LIN {X 104.222,Y 43.174,Z 62.611,A 180.000,B 0.000,C 180.000} C_DIS
LIN {X 104.167,Y 43.026,Z 62.606,A 180.000,B 0.000,C 180.000} C_DIS
LIN {X 104.112,Y 42.878,Z 62.602,A 180.000,B 0.000,C 180.000} C_DIS
LIN {X 104.055,Y 42.732,Z 62.597,A 180.000,B 0.000,C 180.000} C_DIS
LIN {X 103.991,Y 42.588,Z 62.593,A 180.000,B 0.000,C 180.000} C_DIS
LIN {X 103.927,Y 42.444,Z 62.589,A 180.000,B 0.000,C 180.000} C_DIS
LIN {X 103.862,Y 42.300,Z 62.585,A 180.000,B 0.000,C 180.000} C_DIS
LIN {X 103.798,Y 42.156,Z 62.581,A 180.000,B 0.000,C 180.000} C_DIS
LIN {X 103.731,Y 42.014,Z 62.577,A 180.000,B 0.000,C 180.000} C_DIS
LIN {X 103.659,Y 41.874,Z 62.573,A 180.000,B 0.000,C 180.000} C_DIS
LIN {X 103.585,Y 41.735,Z 62.570,A 180.000,B 0.000,C 180.000} C_DIS
LIN {X 103.512,Y 41.595,Z 62.566,A 180.000,B 0.000,C 180.000} C_DIS
LIN {X 103.439,Y 41.456,Z 62.562,A 180.000,B 0.000,C 180.000} C_DIS
LIN {X 103.364,Y 41.317,Z 62.559,A 180.000,B 0.000,C 180.000} C_DIS
LIN {X 103.282,Y 41.183,Z 62.556,A 180.000,B 0.000,C 180.000} C_DIS
LIN {X 103.200,Y 41.048,Z 62.552,A 180.000,B 0.000,C 180.000} C_DIS
LIN {X 103.119,Y 40.913,Z 62.549,A 180.000,B 0.000,C 180.000} C_DIS
LIN {X 103.037,Y 40.779,Z 62.546,A 180.000,B 0.000,C 180.000} C_DIS
LIN {X 102.953,Y 40.646,Z 62.543,A 180.000,B 0.000,C 180.000} C_DIS
LIN {X 102.863,Y 40.516,Z 62.540,A 180.000,B 0.000,C 180.000} C_DIS
LIN {X 102.773,Y 40.387,Z 62.537,A 180.000,B 0.000,C 180.000} C_DIS
LIN {X 102.683,Y 40.258,Z 62.534,A 180.000,B 0.000,C 180.000} C_DIS
LIN {X 102.593,Y 40.128,Z 62.532,A 180.000,B 0.000,C 180.000} C_DIS
LIN {X 102.500,Y 40.001,Z 62.529,A 180.000,B 0.000,C 180.000} C_DIS
LIN {X 102.403,Y 39.878,Z 62.527,A 180.000,B 0.000,C 180.000} C_DIS
LIN {X 102.207,Y 39.631,Z 62.522,A 180.000,B 0.000,C 180.000} C_DIS
LIN {X 102.008,Y 39.386,Z 62.518,A 180.000,B 0.000,C 180.000} C_DIS
LIN {X 101.797,Y 39.152,Z 62.514,A 180.000,B 0.000,C 180.000} C_DIS
LIN {X 101.587,Y 38.918,Z 62.511,A 180.000,B 0.000,C 180.000} C_DIS
LIN {X 101.366,Y 38.694,Z 62.508,A 180.000,B 0.000,C 180.000} C_DIS
LIN {X 101.141,Y 38.473,Z 62.505,A 180.000,B 0.000,C 180.000} C_DIS
LIN {X 100.913,Y 38.256,Z 62.503,A 180.000,B 0.000,C 180.000} C_DIS
LIN {X 100.675,Y 38.050,Z 62.502,A 180.000,B 0.000,C 180.000} C_DIS
LIN {X 100.436,Y 37.844,Z 62.501,A 180.000,B 0.000,C 180.000} C_DIS
LIN {X 100.189,Y 37.649,Z 62.500,A 180.000,B 0.000,C 180.000} C_DIS
LIN {X 100.003,Y 37.508,Z 62.500,A 180.000,B 0.000,C 180.000} C_DIS
; Cutting Move Starts
LIN {X 99.815,Y 37.366,Z 62.500,A 180.000,B 0.000,C 180.000} C_DIS
LIN {X 99.757,Y 37.322,Z 62.500,A 180.000,B 0.000,C 180.000} C_DIS
LIN {X 99.578,Y 37.201,Z 62.500,A 180.000,B 0.000,C 180.000} C_DIS
LIN {X 99.221,Y 36.964,Z 62.500,A 180.000,B 0.000,C 180.000} C_DIS
LIN {X 99.042,Y 36.849,Z 62.500,A 180.000,B 0.000,C 180.000} C_DIS
LIN {X 99.009,Y 36.830,Z 62.500,A 180.000,B 0.000,C 180.000} C_DIS
LIN {X 98.505,Y 36.539,Z 62.500,A 180.000,B 0.000,C 180.000} C_DIS
LIN {X 98.385,Y 36.472,Z 62.500,A 180.000,B 0.000,C 180.000} C_DIS
LIN {X 98.327,Y 36.442,Z 62.500,A 180.000,B 0.000,C 180.000} C_DIS
LIN {X 97.790,Y 36.177,Z 62.500,A 180.000,B 0.000,C 180.000} C_DIS
LIN {X 97.659,Y 36.115,Z 62.500,A 180.000,B 0.000,C 180.000} C_DIS
LIN {X 97.612,Y 36.094,Z 62.500,A 180.000,B 0.000,C 180.000} C_DIS
LIN {X 97.075,Y 35.869,Z 62.500,A 180.000,B 0.000,C 180.000} C_DIS
LIN {X 96.897,Y 35.800,Z 62.500,A 180.000,B 0.000,C 180.000} C_DIS
LIN {X 96.360,Y 35.613,Z 62.500,A 180.000,B 0.000,C 180.000} C_DIS
LIN {X 96.258,Y 35.578,Z 62.500,A 180.000,B 0.000,C 180.000} C_DIS
LIN {X 96.181,Y 35.555,Z 62.500,A 180.000,B 0.000,C 180.000} C_DIS
LIN {X 96.003,Y 35.505,Z 62.500,A 180.000,B 0.000,C 180.000} C_DIS
LIN {X 95.625,Y 35.400,Z 62.500,A 180.000,B 0.000,C 180.000} C_DIS
LIN {X 95.466,Y 35.357,Z 62.500,A 180.000,B 0.000,C 180.000} C_DIS
LIN {X 95.288,Y 35.318,Z 62.500,A 180.000,B 0.000,C 180.000} C_DIS
LIN {X 94.828,Y 35.221,Z 62.500,A 180.000,B 0.000,C 180.000} C_DIS
LIN {X 94.751,Y 35.205,Z 62.500,A 180.000,B 0.000,C 180.000} C_DIS
LIN {X 94.573,Y 35.175,Z 62.500,A 180.000,B 0.000,C 180.000} C_DIS
LIN {X 94.036,Y 35.097,Z 62.500,A 180.000,B 0.000,C 180.000} C_DIS
LIN {X 93.857,Y 35.075,Z 62.500,A 180.000,B 0.000,C 180.000} C_DIS
LIN {X 93.679,Y 35.060,Z 62.500,A 180.000,B 0.000,C 180.000} C_DIS
LIN {X 93.321,Y 35.030,Z 62.500,A 180.000,B 0.000,C 180.000} C_DIS
LIN {X 93.142,Y 35.017,Z 62.500,A 180.000,B 0.000,C 180.000} C_DIS
LIN {X 92.964,Y 35.012,Z 62.500,A 180.000,B 0.000,C 180.000} C_DIS
LIN {X 92.606,Y 35.005,Z 62.500,A 180.000,B 0.000,C 180.000} C_DIS
LIN {X 92.427,Y 35.001,Z 62.500,A 180.000,B 0.000,C 180.000} C_DIS
LIN {X 92.249,Y 35.004,Z 62.500,A 180.000,B 0.000,C 180.000} C_DIS
LIN {X 91.712,Y 35.027,Z 62.500,A 180.000,B 0.000,C 180.000} C_DIS
LIN {X 91.533,Y 35.038,Z 62.500,A 180.000,B 0.000,C 180.000} C_DIS
LIN {X 91.489,Y 35.042,Z 62.500,A 180.000,B 0.000,C 180.000} C_DIS
LIN {X 90.997,Y 35.094,Z 62.500,A 180.000,B 0.000,C 180.000} C_DIS
LIN {X 90.818,Y 35.114,Z 62.500,A 180.000,B 0.000,C 180.000} C_DIS
LIN {X 90.640,Y 35.142,Z 62.500,A 180.000,B 0.000,C 180.000} C_DIS
LIN {X 90.103,Y 35.233,Z 62.500,A 180.000,B 0.000,C 180.000} C_DIS
LIN {X 89.925,Y 35.270,Z 62.500,A 180.000,B 0.000,C 180.000} C_DIS
LIN {X 89.372,Y 35.400,Z 62.500,A 180.000,B 0.000,C 180.000} C_DIS
LIN {X 89.209,Y 35.441,Z 62.500,A 180.000,B 0.000,C 180.000} C_DIS
LIN {X 89.031,Y 35.495,Z 62.500,A 180.000,B 0.000,C 180.000} C_DIS
LIN {X 88.673,Y 35.603,Z 62.500,A 180.000,B 0.000,C 180.000} C_DIS
LIN {X 88.494,Y 35.659,Z 62.500,A 180.000,B 0.000,C 180.000} C_DIS
LIN {X 45.590,Y 50.133,Z 62.500,A 180.000,B 0.000,C 180.000} C_DIS
LIN {X 45.411,Y 50.194,Z 62.500,A 180.000,B 0.000,C 180.000} C_DIS
LIN {X 45.296,Y 50.238,Z 62.500,A 180.000,B 0.000,C 180.000} C_DIS
LIN {X 45.232,Y 50.265,Z 62.500,A 180.000,B 0.000,C 180.000} C_DIS
LIN {X 45.053,Y 50.353,Z 62.500,A 180.000,B 0.000,C 180.000} C_DIS
LIN {X 44.944,Y 50.416,Z 62.500,A 180.000,B 0.000,C 180.000} C_DIS
LIN {X 44.874,Y 50.461,Z 62.500,A 180.000,B 0.000,C 180.000} C_DIS
LIN {X 44.785,Y 50.522,Z 62.500,A 180.000,B 0.000,C 180.000} C_DIS
LIN {X 44.696,Y 50.590,Z 62.500,A 180.000,B 0.000,C 180.000} C_DIS
LIN {X 44.689,Y 50.595,Z 62.500,A 180.000,B 0.000,C 180.000} C_DIS
LIN {X 44.603,Y 50.667,Z 62.500,A 180.000,B 0.000,C 180.000} C_DIS
LIN {X 44.517,Y 50.746,Z 62.500,A 180.000,B 0.000,C 180.000} C_DIS
LIN {X 44.488,Y 50.774,Z 62.500,A 180.000,B 0.000,C 180.000} C_DIS
LIN {X 44.410,Y 50.855,Z 62.500,A 180.000,B 0.000,C 180.000} C_DIS
LIN {X 44.338,Y 50.936,Z 62.500,A 180.000,B 0.000,C 180.000} C_DIS
LIN {X 44.325,Y 50.953,Z 62.500,A 180.000,B 0.000,C 180.000} C_DIS
LIN {X 44.254,Y 51.042,Z 62.500,A 180.000,B 0.000,C 180.000} C_DIS
LIN {X 44.189,Y 51.131,Z 62.500,A 180.000,B 0.000,C 180.000} C_DIS
LIN {X 44.159,Y 51.176,Z 62.500,A 180.000,B 0.000,C 180.000} C_DIS
LIN {X 44.077,Y 51.310,Z 62.500,A 180.000,B 0.000,C 180.000} C_DIS
LIN {X 43.984,Y 51.489,Z 62.500,A 180.000,B 0.000,C 180.000} C_DIS
LIN {X 43.981,Y 51.497,Z 62.500,A 180.000,B 0.000,C 180.000} C_DIS
LIN {X 43.909,Y 51.668,Z 62.500,A 180.000,B 0.000,C 180.000} C_DIS
LIN {X 43.849,Y 51.847,Z 62.500,A 180.000,B 0.000,C 180.000} C_DIS
LIN {X 43.804,Y 52.025,Z 62.500,A 180.000,B 0.000,C 180.000} C_DIS
LIN {X 43.802,Y 52.035,Z 62.500,A 180.000,B 0.000,C 180.000} C_DIS
LIN {X 43.772,Y 52.204,Z 62.500,A 180.000,B 0.000,C 180.000} C_DIS
LIN {X 43.754,Y 52.383,Z 62.500,A 180.000,B 0.000,C 180.000} C_DIS
LIN {X 43.748,Y 52.562,Z 62.500,A 180.000,B 0.000,C 180.000} C_DIS
LIN {X 43.756,Y 52.740,Z 62.500,A 180.000,B 0.000,C 180.000} C_DIS
LIN {X 43.776,Y 52.919,Z 62.500,A 180.000,B 0.000,C 180.000} C_DIS
LIN {X 43.802,Y 53.064,Z 62.500,A 180.000,B 0.000,C 180.000} C_DIS
LIN {X 43.809,Y 53.098,Z 62.500,A 180.000,B 0.000,C 180.000} C_DIS
LIN {X 43.856,Y 53.277,Z 62.500,A 180.000,B 0.000,C 180.000} C_DIS
LIN {X 43.916,Y 53.455,Z 62.500,A 180.000,B 0.000,C 180.000} C_DIS
LIN {X 50.248,Y 72.226,Z 62.500,A 180.000,B 0.000,C 180.000} C_DIS
LIN {X 50.311,Y 72.405,Z 62.500,A 180.000,B 0.000,C 180.000} C_DIS
LIN {X 50.388,Y 72.584,Z 62.500,A 180.000,B 0.000,C 180.000} C_DIS
LIN {X 50.416,Y 72.640,Z 62.500,A 180.000,B 0.000,C 180.000} C_DIS
LIN {X 50.484,Y 72.763,Z 62.500,A 180.000,B 0.000,C 180.000} C_DIS
LIN {X 50.595,Y 72.936,Z 62.500,A 180.000,B 0.000,C 180.000} C_DIS
LIN {X 50.599,Y 72.941,Z 62.500,A 180.000,B 0.000,C 180.000} C_DIS
LIN {X 50.665,Y 73.031,Z 62.500,A 180.000,B 0.000,C 180.000} C_DIS
LIN {X 50.737,Y 73.120,Z 62.500,A 180.000,B 0.000,C 180.000} C_DIS
LIN {X 50.774,Y 73.162,Z 62.500,A 180.000,B 0.000,C 180.000} C_DIS
LIN {X 50.905,Y 73.299,Z 62.500,A 180.000,B 0.000,C 180.000} C_DIS
LIN {X 50.953,Y 73.343,Z 62.500,A 180.000,B 0.000,C 180.000} C_DIS
LIN {X 51.112,Y 73.478,Z 62.500,A 180.000,B 0.000,C 180.000} C_DIS
LIN {X 51.131,Y 73.493,Z 62.500,A 180.000,B 0.000,C 180.000} C_DIS
LIN {X 51.310,Y 73.616,Z 62.500,A 180.000,B 0.000,C 180.000} C_DIS
LIN {X 51.376,Y 73.656,Z 62.500,A 180.000,B 0.000,C 180.000} C_DIS
LIN {X 51.489,Y 73.719,Z 62.500,A 180.000,B 0.000,C 180.000} C_DIS
LIN {X 51.668,Y 73.803,Z 62.500,A 180.000,B 0.000,C 180.000} C_DIS
LIN {X 51.749,Y 73.835,Z 62.500,A 180.000,B 0.000,C 180.000} C_DIS
LIN {X 51.847,Y 73.870,Z 62.500,A 180.000,B 0.000,C 180.000} C_DIS
LIN {X 52.025,Y 73.923,Z 62.500,A 180.000,B 0.000,C 180.000} C_DIS
LIN {X 52.204,Y 73.961,Z 62.500,A 180.000,B 0.000,C 180.000} C_DIS
LIN {X 52.383,Y 73.987,Z 62.500,A 180.000,B 0.000,C 180.000} C_DIS
LIN {X 52.562,Y 73.999,Z 62.500,A 180.000,B 0.000,C 180.000} C_DIS
LIN {X 52.740,Y 73.998,Z 62.500,A 180.000,B 0.000,C 180.000} C_DIS
LIN {X 52.919,Y 73.985,Z 62.500,A 180.000,B 0.000,C 180.000} C_DIS
LIN {X 53.098,Y 73.958,Z 62.500,A 180.000,B 0.000,C 180.000} C_DIS
LIN {X 53.277,Y 73.918,Z 62.500,A 180.000,B 0.000,C 180.000} C_DIS
LIN {X 53.455,Y 73.864,Z 62.500,A 180.000,B 0.000,C 180.000} C_DIS
LIN {X 83.198,Y 63.830,Z 62.500,A 180.000,B 0.000,C 180.000} C_DIS
LIN {X 96.464,Y 59.355,Z 62.500,A 180.000,B 0.000,C 180.000} C_DIS
LIN {X 96.539,Y 59.329,Z 62.500,A 180.000,B 0.000,C 180.000} C_DIS
LIN {X 96.718,Y 59.263,Z 62.500,A 180.000,B 0.000,C 180.000} C_DIS
LIN {X 97.075,Y 59.129,Z 62.500,A 180.000,B 0.000,C 180.000} C_DIS
LIN {X 97.254,Y 59.061,Z 62.500,A 180.000,B 0.000,C 180.000} C_DIS
LIN {X 97.397,Y 58.997,Z 62.500,A 180.000,B 0.000,C 180.000} C_DIS
LIN {X 97.798,Y 58.819,Z 62.500,A 180.000,B 0.000,C 180.000} C_DIS
LIN {X 97.969,Y 58.740,Z 62.500,A 180.000,B 0.000,C 180.000} C_DIS
LIN {X 98.148,Y 58.647,Z 62.500,A 180.000,B 0.000,C 180.000} C_DIS
LIN {X 98.505,Y 58.460,Z 62.500,A 180.000,B 0.000,C 180.000} C_DIS
LIN {X 98.684,Y 58.363,Z 62.500,A 180.000,B 0.000,C 180.000} C_DIS
LIN {X 98.817,Y 58.282,Z 62.500,A 180.000,B 0.000,C 180.000} C_DIS
LIN {X 99.221,Y 58.038,Z 62.500,A 180.000,B 0.000,C 180.000} C_DIS
LIN {X 99.395,Y 57.925,Z 62.500,A 180.000,B 0.000,C 180.000} C_DIS
LIN {X 99.757,Y 57.673,Z 62.500,A 180.000,B 0.000,C 180.000} C_DIS
LIN {X 99.909,Y 57.567,Z 62.500,A 180.000,B 0.000,C 180.000} C_DIS
LIN {X 99.936,Y 57.548,Z 62.500,A 180.000,B 0.000,C 180.000} C_DIS
LIN {X 100.114,Y 57.409,Z 62.500,A 180.000,B 0.000,C 180.000} C_DIS
LIN {X 100.472,Y 57.125,Z 62.500,A 180.000,B 0.000,C 180.000} C_DIS
LIN {X 100.588,Y 57.031,Z 62.500,A 180.000,B 0.000,C 180.000} C_DIS
LIN {X 100.651,Y 56.975,Z 62.500,A 180.000,B 0.000,C 180.000} C_DIS
LIN {X 101.008,Y 56.653,Z 62.500,A 180.000,B 0.000,C 180.000} C_DIS
LIN {X 101.180,Y 56.495,Z 62.500,A 180.000,B 0.000,C 180.000} C_DIS
LIN {X 101.187,Y 56.488,Z 62.500,A 180.000,B 0.000,C 180.000} C_DIS
LIN {X 101.356,Y 56.316,Z 62.500,A 180.000,B 0.000,C 180.000} C_DIS
LIN {X 101.545,Y 56.123,Z 62.500,A 180.000,B 0.000,C 180.000} C_DIS
LIN {X 101.704,Y 55.958,Z 62.500,A 180.000,B 0.000,C 180.000} C_DIS
LIN {X 101.723,Y 55.937,Z 62.500,A 180.000,B 0.000,C 180.000} C_DIS
LIN {X 101.860,Y 55.779,Z 62.500,A 180.000,B 0.000,C 180.000} C_DIS
LIN {X 102.168,Y 55.422,Z 62.500,A 180.000,B 0.000,C 180.000} C_DIS
LIN {X 102.260,Y 55.309,Z 62.500,A 180.000,B 0.000,C 180.000} C_DIS
LIN {X 102.310,Y 55.243,Z 62.500,A 180.000,B 0.000,C 180.000} C_DIS
LIN {X 102.617,Y 54.837,Z 62.500,A 180.000,B 0.000,C 180.000} C_DIS
LIN {X 102.713,Y 54.707,Z 62.500,A 180.000,B 0.000,C 180.000} C_DIS
LIN {X 102.796,Y 54.583,Z 62.500,A 180.000,B 0.000,C 180.000} C_DIS
LIN {X 103.069,Y 54.171,Z 62.500,A 180.000,B 0.000,C 180.000} C_DIS
LIN {X 103.153,Y 54.038,Z 62.500,A 180.000,B 0.000,C 180.000} C_DIS
LIN {X 103.180,Y 53.992,Z 62.500,A 180.000,B 0.000,C 180.000} C_DIS
LIN {X 103.386,Y 53.634,Z 62.500,A 180.000,B 0.000,C 180.000} C_DIS
LIN {X 103.489,Y 53.455,Z 62.500,A 180.000,B 0.000,C 180.000} C_DIS
LIN {X 103.511,Y 53.417,Z 62.500,A 180.000,B 0.000,C 180.000} C_DIS
LIN {X 103.583,Y 53.277,Z 62.500,A 180.000,B 0.000,C 180.000} C_DIS
LIN {X 103.760,Y 52.919,Z 62.500,A 180.000,B 0.000,C 180.000} C_DIS
LIN {X 103.848,Y 52.740,Z 62.500,A 180.000,B 0.000,C 180.000} C_DIS
LIN {X 103.869,Y 52.697,Z 62.500,A 180.000,B 0.000,C 180.000} C_DIS
LIN {X 103.927,Y 52.562,Z 62.500,A 180.000,B 0.000,C 180.000} C_DIS
LIN {X 104.077,Y 52.204,Z 62.500,A 180.000,B 0.000,C 180.000} C_DIS
LIN {X 104.152,Y 52.025,Z 62.500,A 180.000,B 0.000,C 180.000} C_DIS
LIN {X 104.218,Y 51.847,Z 62.500,A 180.000,B 0.000,C 180.000} C_DIS
LIN {X 104.405,Y 51.307,Z 62.500,A 180.000,B 0.000,C 180.000} C_DIS
LIN {X 104.459,Y 51.131,Z 62.500,A 180.000,B 0.000,C 180.000} C_DIS
LIN {X 104.609,Y 50.595,Z 62.500,A 180.000,B 0.000,C 180.000} C_DIS
LIN {X 104.654,Y 50.416,Z 62.500,A 180.000,B 0.000,C 180.000} C_DIS
LIN {X 104.692,Y 50.238,Z 62.500,A 180.000,B 0.000,C 180.000} C_DIS
LIN {X 104.768,Y 49.880,Z 62.500,A 180.000,B 0.000,C 180.000} C_DIS
LIN {X 104.805,Y 49.701,Z 62.500,A 180.000,B 0.000,C 180.000} C_DIS
LIN {X 104.832,Y 49.523,Z 62.500,A 180.000,B 0.000,C 180.000} C_DIS
LIN {X 104.885,Y 49.165,Z 62.500,A 180.000,B 0.000,C 180.000} C_DIS
LIN {X 104.911,Y 48.986,Z 62.500,A 180.000,B 0.000,C 180.000} C_DIS
LIN {X 104.929,Y 48.807,Z 62.500,A 180.000,B 0.000,C 180.000} C_DIS
LIN {X 104.974,Y 48.271,Z 62.500,A 180.000,B 0.000,C 180.000} C_DIS
LIN {X 104.986,Y 48.092,Z 62.500,A 180.000,B 0.000,C 180.000} C_DIS
LIN {X 104.989,Y 47.914,Z 62.500,A 180.000,B 0.000,C 180.000} C_DIS
LIN {X 104.996,Y 47.556,Z 62.500,A 180.000,B 0.000,C 180.000} C_DIS
LIN {X 104.999,Y 47.377,Z 62.500,A 180.000,B 0.000,C 180.000} C_DIS
LIN {X 104.994,Y 47.198,Z 62.500,A 180.000,B 0.000,C 180.000} C_DIS
LIN {X 104.971,Y 46.662,Z 62.500,A 180.000,B 0.000,C 180.000} C_DIS
LIN {X 104.957,Y 46.483,Z 62.500,A 180.000,B 0.000,C 180.000} C_DIS
LIN {X 104.900,Y 45.947,Z 62.500,A 180.000,B 0.000,C 180.000} C_DIS
LIN {X 104.879,Y 45.768,Z 62.500,A 180.000,B 0.000,C 180.000} C_DIS
LIN {X 104.850,Y 45.590,Z 62.500,A 180.000,B 0.000,C 180.000} C_DIS
LIN {X 104.789,Y 45.232,Z 62.500,A 180.000,B 0.000,C 180.000} C_DIS
LIN {X 104.762,Y 45.077,Z 62.500,A 180.000,B 0.000,C 180.000} C_DIS
LIN {X 104.758,Y 45.053,Z 62.500,A 180.000,B 0.000,C 180.000} C_DIS
LIN {X 104.719,Y 44.874,Z 62.500,A 180.000,B 0.000,C 180.000} C_DIS
LIN {X 104.592,Y 44.338,Z 62.500,A 180.000,B 0.000,C 180.000} C_DIS
LIN {X 104.584,Y 44.302,Z 62.500,A 180.000,B 0.000,C 180.000} C_DIS
LIN {X 104.544,Y 44.159,Z 62.500,A 180.000,B 0.000,C 180.000} C_DIS
LIN {X 104.381,Y 43.623,Z 62.500,A 180.000,B 0.000,C 180.000} C_DIS
LIN {X 104.323,Y 43.444,Z 62.500,A 180.000,B 0.000,C 180.000} C_DIS
LIN {X 104.257,Y 43.266,Z 62.500,A 180.000,B 0.000,C 180.000} C_DIS
LIN {X 104.123,Y 42.908,Z 62.500,A 180.000,B 0.000,C 180.000} C_DIS
LIN {X 104.053,Y 42.729,Z 62.500,A 180.000,B 0.000,C 180.000} C_DIS
LIN {X 104.047,Y 42.715,Z 62.500,A 180.000,B 0.000,C 180.000} C_DIS
LIN {X 103.974,Y 42.550,Z 62.500,A 180.000,B 0.000,C 180.000} C_DIS
LIN {X 103.814,Y 42.193,Z 62.500,A 180.000,B 0.000,C 180.000} C_DIS
LIN {X 103.732,Y 42.014,Z 62.500,A 180.000,B 0.000,C 180.000} C_DIS
LIN {X 103.690,Y 41.934,Z 62.500,A 180.000,B 0.000,C 180.000} C_DIS
LIN {X 103.451,Y 41.478,Z 62.500,A 180.000,B 0.000,C 180.000} C_DIS
LIN {X 103.353,Y 41.299,Z 62.500,A 180.000,B 0.000,C 180.000} C_DIS
LIN {X 103.332,Y 41.265,Z 62.500,A 180.000,B 0.000,C 180.000} C_DIS
LIN {X 103.027,Y 40.763,Z 62.500,A 180.000,B 0.000,C 180.000} C_DIS
LIN {X 102.975,Y 40.679,Z 62.500,A 180.000,B 0.000,C 180.000} C_DIS
LIN {X 102.910,Y 40.584,Z 62.500,A 180.000,B 0.000,C 180.000} C_DIS
LIN {X 102.617,Y 40.163,Z 62.500,A 180.000,B 0.000,C 180.000} C_DIS
LIN {X 102.536,Y 40.048,Z 62.500,A 180.000,B 0.000,C 180.000} C_DIS
LIN {X 102.438,Y 39.923,Z 62.500,A 180.000,B 0.000,C 180.000} C_DIS
LIN {X 102.112,Y 39.511,Z 62.500,A 180.000,B 0.000,C 180.000} C_DIS
LIN {X 102.081,Y 39.472,Z 62.500,A 180.000,B 0.000,C 180.000} C_DIS
LIN {X 101.960,Y 39.333,Z 62.500,A 180.000,B 0.000,C 180.000} C_DIS
LIN {X 101.638,Y 38.975,Z 62.500,A 180.000,B 0.000,C 180.000} C_DIS
LIN {X 101.545,Y 38.872,Z 62.500,A 180.000,B 0.000,C 180.000} C_DIS
LIN {X 101.471,Y 38.796,Z 62.500,A 180.000,B 0.000,C 180.000} C_DIS
LIN {X 101.366,Y 38.693,Z 62.500,A 180.000,B 0.000,C 180.000} C_DIS
LIN {X 101.008,Y 38.344,Z 62.500,A 180.000,B 0.000,C 180.000} C_DIS
LIN {X 100.918,Y 38.260,Z 62.500,A 180.000,B 0.000,C 180.000} C_DIS
LIN {X 100.829,Y 38.183,Z 62.500,A 180.000,B 0.000,C 180.000} C_DIS
LIN {X 100.472,Y 37.875,Z 62.500,A 180.000,B 0.000,C 180.000} C_DIS
LIN {X 100.293,Y 37.728,Z 62.500,A 180.000,B 0.000,C 180.000} C_DIS
LIN {X 100.003,Y 37.508,Z 62.500,A 180.000,B 0.000,C 180.000} C_DIS
; Link Move Starts
LIN {X 99.752,Y 37.319,Z 62.500,A 180.000,B 0.000,C 180.000} C_DIS
LIN {X 99.490,Y 37.143,Z 62.498,A 180.000,B 0.000,C 180.000} C_DIS
LIN {X 99.228,Y 36.969,Z 62.496,A 180.000,B 0.000,C 180.000} C_DIS
LIN {X 98.961,Y 36.802,Z 62.492,A 180.000,B 0.000,C 180.000} C_DIS
LIN {X 98.688,Y 36.645,Z 62.488,A 180.000,B 0.000,C 180.000} C_DIS
LIN {X 98.415,Y 36.488,Z 62.483,A 180.000,B 0.000,C 180.000} C_DIS
LIN {X 98.274,Y 36.416,Z 62.481,A 180.000,B 0.000,C 180.000} C_DIS
LIN {X 98.133,Y 36.346,Z 62.478,A 180.000,B 0.000,C 180.000} C_DIS
LIN {X 97.992,Y 36.276,Z 62.475,A 180.000,B 0.000,C 180.000} C_DIS
LIN {X 97.851,Y 36.207,Z 62.471,A 180.000,B 0.000,C 180.000} C_DIS
LIN {X 97.709,Y 36.137,Z 62.468,A 180.000,B 0.000,C 180.000} C_DIS
LIN {X 97.565,Y 36.075,Z 62.464,A 180.000,B 0.000,C 180.000} C_DIS
LIN {X 97.420,Y 36.014,Z 62.460,A 180.000,B 0.000,C 180.000} C_DIS
LIN {X 97.274,Y 35.953,Z 62.456,A 180.000,B 0.000,C 180.000} C_DIS
LIN {X 97.129,Y 35.892,Z 62.452,A 180.000,B 0.000,C 180.000} C_DIS
LIN {X 96.984,Y 35.832,Z 62.448,A 180.000,B 0.000,C 180.000} C_DIS
LIN {X 96.835,Y 35.779,Z 62.444,A 180.000,B 0.000,C 180.000} C_DIS
LIN {X 96.687,Y 35.727,Z 62.439,A 180.000,B 0.000,C 180.000} C_DIS
LIN {X 96.538,Y 35.675,Z 62.434,A 180.000,B 0.000,C 180.000} C_DIS
LIN {X 96.389,Y 35.623,Z 62.429,A 180.000,B 0.000,C 180.000} C_DIS
LIN {X 96.240,Y 35.573,Z 62.424,A 180.000,B 0.000,C 180.000} C_DIS
LIN {X 96.165,Y 35.550,Z 62.422,A 180.000,B 0.000,C 180.000} C_DIS
LIN {X 96.089,Y 35.529,Z 62.419,A 180.000,B 0.000,C 180.000} C_DIS
LIN {X 96.013,Y 35.508,Z 62.417,A 180.000,B 0.000,C 180.000} C_DIS
LIN {X 95.937,Y 35.487,Z 62.414,A 180.000,B 0.000,C 180.000} C_DIS
LIN {X 95.861,Y 35.465,Z 62.411,A 180.000,B 0.000,C 180.000} C_DIS
LIN {X 95.785,Y 35.444,Z 62.409,A 180.000,B 0.000,C 180.000} C_DIS
LIN {X 95.709,Y 35.423,Z 62.406,A 180.000,B 0.000,C 180.000} C_DIS
LIN {X 95.634,Y 35.402,Z 62.403,A 180.000,B 0.000,C 180.000} C_DIS
LIN {X 95.558,Y 35.381,Z 62.401,A 180.000,B 0.000,C 180.000} C_DIS
LIN {X 95.482,Y 35.361,Z 62.398,A 180.000,B 0.000,C 180.000} C_DIS
LIN {X 95.405,Y 35.343,Z 62.395,A 180.000,B 0.000,C 180.000} C_DIS
LIN {X 95.328,Y 35.327,Z 62.392,A 180.000,B 0.000,C 180.000} C_DIS
LIN {X 95.251,Y 35.310,Z 62.389,A 180.000,B 0.000,C 180.000} C_DIS
LIN {X 95.174,Y 35.294,Z 62.387,A 180.000,B 0.000,C 180.000} C_DIS
LIN {X 95.097,Y 35.278,Z 62.384,A 180.000,B 0.000,C 180.000} C_DIS
LIN {X 95.020,Y 35.261,Z 62.381,A 180.000,B 0.000,C 180.000} C_DIS
LIN {X 94.943,Y 35.245,Z 62.378,A 180.000,B 0.000,C 180.000} C_DIS
LIN {X 94.866,Y 35.229,Z 62.376,A 180.000,B 0.000,C 180.000} C_DIS
LIN {X 94.788,Y 35.212,Z 62.373,A 180.000,B 0.000,C 180.000} C_DIS
LIN {X 94.711,Y 35.197,Z 62.370,A 180.000,B 0.000,C 180.000} C_DIS
LIN {X 94.634,Y 35.184,Z 62.367,A 180.000,B 0.000,C 180.000} C_DIS
LIN {X 94.556,Y 35.173,Z 62.365,A 180.000,B 0.000,C 180.000} C_DIS
LIN {X 94.478,Y 35.161,Z 62.362,A 180.000,B 0.000,C 180.000} C_DIS
LIN {X 94.322,Y 35.138,Z 62.356,A 180.000,B 0.000,C 180.000} C_DIS
LIN {X 94.244,Y 35.127,Z 62.354,A 180.000,B 0.000,C 180.000} C_DIS
LIN {X 94.088,Y 35.104,Z 62.348,A 180.000,B 0.000,C 180.000} C_DIS
LIN {X 94.010,Y 35.093,Z 62.345,A 180.000,B 0.000,C 180.000} C_DIS
LIN {X 93.932,Y 35.082,Z 62.343,A 180.000,B 0.000,C 180.000} C_DIS
LIN {X 93.854,Y 35.074,Z 62.340,A 180.000,B 0.000,C 180.000} C_DIS
LIN {X 93.697,Y 35.061,Z 62.334,A 180.000,B 0.000,C 180.000} C_DIS
LIN {X 93.618,Y 35.055,Z 62.332,A 180.000,B 0.000,C 180.000} C_DIS
LIN {X 93.461,Y 35.042,Z 62.326,A 180.000,B 0.000,C 180.000} C_DIS
LIN {X 93.226,Y 35.022,Z 62.318,A 180.000,B 0.000,C 180.000} C_DIS
LIN {X 93.147,Y 35.017,Z 62.315,A 180.000,B 0.000,C 180.000} C_DIS
LIN {X 93.069,Y 35.014,Z 62.312,A 180.000,B 0.000,C 180.000} C_DIS
LIN {X 92.990,Y 35.012,Z 62.310,A 180.000,B 0.000,C 180.000} C_DIS
LIN {X 92.832,Y 35.009,Z 62.304,A 180.000,B 0.000,C 180.000} C_DIS
LIN {X 92.439,Y 35.001,Z 62.290,A 180.000,B 0.000,C 180.000} C_DIS
LIN {X 92.360,Y 35.001,Z 62.288,A 180.000,B 0.000,C 180.000} C_DIS
LIN {X 92.281,Y 35.003,Z 62.285,A 180.000,B 0.000,C 180.000} C_DIS
LIN {X 91.809,Y 35.023,Z 62.268,A 180.000,B 0.000,C 180.000} C_DIS
LIN {X 91.652,Y 35.030,Z 62.263,A 180.000,B 0.000,C 180.000} C_DIS
LIN {X 91.573,Y 35.034,Z 62.260,A 180.000,B 0.000,C 180.000} C_DIS
LIN {X 91.495,Y 35.042,Z 62.257,A 180.000,B 0.000,C 180.000} C_DIS
LIN {X 90.868,Y 35.108,Z 62.235,A 180.000,B 0.000,C 180.000} C_DIS
LIN {X 90.790,Y 35.117,Z 62.233,A 180.000,B 0.000,C 180.000} C_DIS
LIN {X 90.712,Y 35.130,Z 62.230,A 180.000,B 0.000,C 180.000} C_DIS
LIN {X 90.091,Y 35.235,Z 62.208,A 180.000,B 0.000,C 180.000} C_DIS
LIN {X 90.014,Y 35.250,Z 62.205,A 180.000,B 0.000,C 180.000} C_DIS
LIN {X 89.937,Y 35.267,Z 62.202,A 180.000,B 0.000,C 180.000} C_DIS
LIN {X 89.860,Y 35.285,Z 62.200,A 180.000,B 0.000,C 180.000} C_DIS
LIN {X 89.707,Y 35.321,Z 62.194,A 180.000,B 0.000,C 180.000} C_DIS
LIN {X 89.400,Y 35.393,Z 62.183,A 180.000,B 0.000,C 180.000} C_DIS
LIN {X 89.324,Y 35.411,Z 62.180,A 180.000,B 0.000,C 180.000} C_DIS
LIN {X 89.247,Y 35.431,Z 62.178,A 180.000,B 0.000,C 180.000} C_DIS
LIN {X 89.172,Y 35.452,Z 62.175,A 180.000,B 0.000,C 180.000} C_DIS
LIN {X 89.021,Y 35.498,Z 62.169,A 180.000,B 0.000,C 180.000} C_DIS
LIN {X 88.946,Y 35.521,Z 62.167,A 180.000,B 0.000,C 180.000} C_DIS
LIN {X 88.795,Y 35.567,Z 62.161,A 180.000,B 0.000,C 180.000} C_DIS
LIN {X 88.644,Y 35.612,Z 62.156,A 180.000,B 0.000,C 180.000} C_DIS
LIN {X 88.569,Y 35.635,Z 62.153,A 180.000,B 0.000,C 180.000} C_DIS
LIN {X 88.494,Y 35.659,Z 62.150,A 180.000,B 0.000,C 180.000} C_DIS
LIN {X 88.345,Y 35.710,Z 62.145,A 180.000,B 0.000,C 180.000} C_DIS
LIN {X 88.195,Y 35.760,Z 62.139,A 180.000,B 0.000,C 180.000} C_DIS
LIN {X 88.121,Y 35.785,Z 62.136,A 180.000,B 0.000,C 180.000} C_DIS
LIN {X 88.046,Y 35.810,Z 62.134,A 180.000,B 0.000,C 180.000} C_DIS
LIN {X 87.972,Y 35.836,Z 62.131,A 180.000,B 0.000,C 180.000} C_DIS
LIN {X 87.897,Y 35.861,Z 62.128,A 180.000,B 0.000,C 180.000} C_DIS
LIN {X 87.822,Y 35.886,Z 62.125,A 180.000,B 0.000,C 180.000} C_DIS
LIN {X 87.748,Y 35.911,Z 62.123,A 180.000,B 0.000,C 180.000} C_DIS
LIN {X 87.673,Y 35.936,Z 62.120,A 180.000,B 0.000,C 180.000} C_DIS
LIN {X 87.598,Y 35.961,Z 62.117,A 180.000,B 0.000,C 180.000} C_DIS
LIN {X 87.524,Y 35.987,Z 62.114,A 180.000,B 0.000,C 180.000} C_DIS
LIN {X 87.449,Y 36.012,Z 62.112,A 180.000,B 0.000,C 180.000} C_DIS
LIN {X 87.375,Y 36.037,Z 62.109,A 180.000,B 0.000,C 180.000} C_DIS
LIN {X 87.300,Y 36.062,Z 62.106,A 180.000,B 0.000,C 180.000} C_DIS
LIN {X 87.225,Y 36.087,Z 62.103,A 180.000,B 0.000,C 180.000} C_DIS
LIN {X 87.151,Y 36.112,Z 62.101,A 180.000,B 0.000,C 180.000} C_DIS
LIN {X 87.076,Y 36.138,Z 62.098,A 180.000,B 0.000,C 180.000} C_DIS
LIN {X 87.002,Y 36.163,Z 62.095,A 180.000,B 0.000,C 180.000} C_DIS
LIN {X 86.927,Y 36.188,Z 62.092,A 180.000,B 0.000,C 180.000} C_DIS
LIN {X 86.852,Y 36.213,Z 62.090,A 180.000,B 0.000,C 180.000} C_DIS
LIN {X 86.778,Y 36.238,Z 62.087,A 180.000,B 0.000,C 180.000} C_DIS
LIN {X 86.703,Y 36.263,Z 62.084,A 180.000,B 0.000,C 180.000} C_DIS
LIN {X 86.628,Y 36.289,Z 62.082,A 180.000,B 0.000,C 180.000} C_DIS
LIN {X 86.554,Y 36.314,Z 62.079,A 180.000,B 0.000,C 180.000} C_DIS
LIN {X 86.479,Y 36.339,Z 62.077,A 180.000,B 0.000,C 180.000} C_DIS
LIN {X 86.405,Y 36.364,Z 62.074,A 180.000,B 0.000,C 180.000} C_DIS
LIN {X 86.255,Y 36.415,Z 62.069,A 180.000,B 0.000,C 180.000} C_DIS
LIN {X 86.106,Y 36.465,Z 62.064,A 180.000,B 0.000,C 180.000} C_DIS
LIN {X 85.957,Y 36.515,Z 62.060,A 180.000,B 0.000,C 180.000} C_DIS
LIN {X 85.808,Y 36.566,Z 62.055,A 180.000,B 0.000,C 180.000} C_DIS
LIN {X 85.658,Y 36.616,Z 62.051,A 180.000,B 0.000,C 180.000} C_DIS
LIN {X 85.509,Y 36.666,Z 62.047,A 180.000,B 0.000,C 180.000} C_DIS
LIN {X 85.360,Y 36.717,Z 62.042,A 180.000,B 0.000,C 180.000} C_DIS
LIN {X 85.211,Y 36.767,Z 62.039,A 180.000,B 0.000,C 180.000} C_DIS
LIN {X 85.061,Y 36.817,Z 62.035,A 180.000,B 0.000,C 180.000} C_DIS
LIN {X 84.912,Y 36.868,Z 62.031,A 180.000,B 0.000,C 180.000} C_DIS
LIN {X 84.763,Y 36.918,Z 62.028,A 180.000,B 0.000,C 180.000} C_DIS
LIN {X 84.614,Y 36.968,Z 62.024,A 180.000,B 0.000,C 180.000} C_DIS
LIN {X 84.465,Y 37.019,Z 62.021,A 180.000,B 0.000,C 180.000} C_DIS
LIN {X 84.315,Y 37.069,Z 62.019,A 180.000,B 0.000,C 180.000} C_DIS
LIN {X 84.166,Y 37.119,Z 62.016,A 180.000,B 0.000,C 180.000} C_DIS
LIN {X 83.868,Y 37.220,Z 62.011,A 180.000,B 0.000,C 180.000} C_DIS
LIN {X 83.569,Y 37.321,Z 62.007,A 180.000,B 0.000,C 180.000} C_DIS
LIN {X 83.271,Y 37.421,Z 62.004,A 180.000,B 0.000,C 180.000} C_DIS
LIN {X 82.972,Y 37.522,Z 62.002,A 180.000,B 0.000,C 180.000} C_DIS
LIN {X 82.674,Y 37.623,Z 62.000,A 180.000,B 0.000,C 180.000} C_DIS
LIN {X 82.417,Y 37.709,Z 62.000,A 180.000,B 0.000,C 180.000} C_DIS
; Cutting Move Starts
LIN {X 45.590,Y 50.133,Z 62.000,A 180.000,B 0.000,C 180.000} C_DIS
LIN {X 45.411,Y 50.194,Z 62.000,A 180.000,B 0.000,C 180.000} C_DIS
LIN {X 45.296,Y 50.238,Z 62.000,A 180.000,B 0.000,C 180.000} C_DIS
LIN {X 45.232,Y 50.265,Z 62.000,A 180.000,B 0.000,C 180.000} C_DIS
LIN {X 45.053,Y 50.353,Z 62.000,A 180.000,B 0.000,C 180.000} C_DIS
LIN {X 44.944,Y 50.416,Z 62.000,A 180.000,B 0.000,C 180.000} C_DIS
LIN {X 44.874,Y 50.461,Z 62.000,A 180.000,B 0.000,C 180.000} C_DIS
LIN {X 44.785,Y 50.522,Z 62.000,A 180.000,B 0.000,C 180.000} C_DIS
LIN {X 44.696,Y 50.590,Z 62.000,A 180.000,B 0.000,C 180.000} C_DIS
LIN {X 44.689,Y 50.595,Z 62.000,A 180.000,B 0.000,C 180.000} C_DIS
LIN {X 44.603,Y 50.667,Z 62.000,A 180.000,B 0.000,C 180.000} C_DIS
LIN {X 44.517,Y 50.746,Z 62.000,A 180.000,B 0.000,C 180.000} C_DIS
LIN {X 44.488,Y 50.774,Z 62.000,A 180.000,B 0.000,C 180.000} C_DIS
LIN {X 44.410,Y 50.855,Z 62.000,A 180.000,B 0.000,C 180.000} C_DIS
LIN {X 44.338,Y 50.936,Z 62.000,A 180.000,B 0.000,C 180.000} C_DIS
LIN {X 44.325,Y 50.953,Z 62.000,A 180.000,B 0.000,C 180.000} C_DIS
LIN {X 44.254,Y 51.042,Z 62.000,A 180.000,B 0.000,C 180.000} C_DIS
LIN {X 44.189,Y 51.131,Z 62.000,A 180.000,B 0.000,C 180.000} C_DIS
LIN {X 44.159,Y 51.176,Z 62.000,A 180.000,B 0.000,C 180.000} C_DIS
LIN {X 44.077,Y 51.310,Z 62.000,A 180.000,B 0.000,C 180.000} C_DIS
LIN {X 43.984,Y 51.489,Z 62.000,A 180.000,B 0.000,C 180.000} C_DIS
LIN {X 43.981,Y 51.497,Z 62.000,A 180.000,B 0.000,C 180.000} C_DIS
LIN {X 43.909,Y 51.668,Z 62.000,A 180.000,B 0.000,C 180.000} C_DIS
LIN {X 43.849,Y 51.847,Z 62.000,A 180.000,B 0.000,C 180.000} C_DIS
LIN {X 43.804,Y 52.025,Z 62.000,A 180.000,B 0.000,C 180.000} C_DIS
LIN {X 43.802,Y 52.035,Z 62.000,A 180.000,B 0.000,C 180.000} C_DIS
LIN {X 43.772,Y 52.204,Z 62.000,A 180.000,B 0.000,C 180.000} C_DIS
LIN {X 43.754,Y 52.383,Z 62.000,A 180.000,B 0.000,C 180.000} C_DIS
LIN {X 43.748,Y 52.562,Z 62.000,A 180.000,B 0.000,C 180.000} C_DIS
LIN {X 43.756,Y 52.740,Z 62.000,A 180.000,B 0.000,C 180.000} C_DIS
LIN {X 43.776,Y 52.919,Z 62.000,A 180.000,B 0.000,C 180.000} C_DIS
LIN {X 43.802,Y 53.064,Z 62.000,A 180.000,B 0.000,C 180.000} C_DIS
LIN {X 43.809,Y 53.098,Z 62.000,A 180.000,B 0.000,C 180.000} C_DIS
LIN {X 43.856,Y 53.277,Z 62.000,A 180.000,B 0.000,C 180.000} C_DIS
LIN {X 43.916,Y 53.455,Z 62.000,A 180.000,B 0.000,C 180.000} C_DIS
LIN {X 50.248,Y 72.226,Z 62.000,A 180.000,B 0.000,C 180.000} C_DIS
LIN {X 50.311,Y 72.405,Z 62.000,A 180.000,B 0.000,C 180.000} C_DIS
LIN {X 50.388,Y 72.584,Z 62.000,A 180.000,B 0.000,C 180.000} C_DIS
LIN {X 50.416,Y 72.640,Z 62.000,A 180.000,B 0.000,C 180.000} C_DIS
LIN {X 50.484,Y 72.763,Z 62.000,A 180.000,B 0.000,C 180.000} C_DIS
LIN {X 50.595,Y 72.936,Z 62.000,A 180.000,B 0.000,C 180.000} C_DIS
LIN {X 50.599,Y 72.941,Z 62.000,A 180.000,B 0.000,C 180.000} C_DIS
LIN {X 50.665,Y 73.031,Z 62.000,A 180.000,B 0.000,C 180.000} C_DIS
LIN {X 50.737,Y 73.120,Z 62.000,A 180.000,B 0.000,C 180.000} C_DIS
LIN {X 50.774,Y 73.162,Z 62.000,A 180.000,B 0.000,C 180.000} C_DIS
LIN {X 50.905,Y 73.299,Z 62.000,A 180.000,B 0.000,C 180.000} C_DIS
LIN {X 50.953,Y 73.343,Z 62.000,A 180.000,B 0.000,C 180.000} C_DIS
LIN {X 51.112,Y 73.478,Z 62.000,A 180.000,B 0.000,C 180.000} C_DIS
LIN {X 51.131,Y 73.493,Z 62.000,A 180.000,B 0.000,C 180.000} C_DIS
LIN {X 51.310,Y 73.616,Z 62.000,A 180.000,B 0.000,C 180.000} C_DIS
LIN {X 51.376,Y 73.656,Z 62.000,A 180.000,B 0.000,C 180.000} C_DIS
LIN {X 51.489,Y 73.719,Z 62.000,A 180.000,B 0.000,C 180.000} C_DIS
LIN {X 51.668,Y 73.803,Z 62.000,A 180.000,B 0.000,C 180.000} C_DIS
LIN {X 51.749,Y 73.835,Z 62.000,A 180.000,B 0.000,C 180.000} C_DIS
LIN {X 51.847,Y 73.870,Z 62.000,A 180.000,B 0.000,C 180.000} C_DIS
LIN {X 52.025,Y 73.923,Z 62.000,A 180.000,B 0.000,C 180.000} C_DIS
LIN {X 52.204,Y 73.961,Z 62.000,A 180.000,B 0.000,C 180.000} C_DIS
LIN {X 52.383,Y 73.987,Z 62.000,A 180.000,B 0.000,C 180.000} C_DIS
LIN {X 52.562,Y 73.999,Z 62.000,A 180.000,B 0.000,C 180.000} C_DIS
LIN {X 52.740,Y 73.998,Z 62.000,A 180.000,B 0.000,C 180.000} C_DIS
LIN {X 52.919,Y 73.985,Z 62.000,A 180.000,B 0.000,C 180.000} C_DIS
LIN {X 53.098,Y 73.958,Z 62.000,A 180.000,B 0.000,C 180.000} C_DIS
LIN {X 53.277,Y 73.918,Z 62.000,A 180.000,B 0.000,C 180.000} C_DIS
LIN {X 53.455,Y 73.864,Z 62.000,A 180.000,B 0.000,C 180.000} C_DIS
LIN {X 83.198,Y 63.830,Z 62.000,A 180.000,B 0.000,C 180.000} C_DIS
LIN {X 96.464,Y 59.355,Z 62.000,A 180.000,B 0.000,C 180.000} C_DIS
LIN {X 96.539,Y 59.329,Z 62.000,A 180.000,B 0.000,C 180.000} C_DIS
LIN {X 96.718,Y 59.263,Z 62.000,A 180.000,B 0.000,C 180.000} C_DIS
LIN {X 97.075,Y 59.129,Z 62.000,A 180.000,B 0.000,C 180.000} C_DIS
LIN {X 97.254,Y 59.061,Z 62.000,A 180.000,B 0.000,C 180.000} C_DIS
LIN {X 97.397,Y 58.997,Z 62.000,A 180.000,B 0.000,C 180.000} C_DIS
LIN {X 97.798,Y 58.819,Z 62.000,A 180.000,B 0.000,C 180.000} C_DIS
LIN {X 97.969,Y 58.740,Z 62.000,A 180.000,B 0.000,C 180.000} C_DIS
LIN {X 98.148,Y 58.647,Z 62.000,A 180.000,B 0.000,C 180.000} C_DIS
LIN {X 98.505,Y 58.460,Z 62.000,A 180.000,B 0.000,C 180.000} C_DIS
LIN {X 98.684,Y 58.363,Z 62.000,A 180.000,B 0.000,C 180.000} C_DIS
LIN {X 98.817,Y 58.282,Z 62.000,A 180.000,B 0.000,C 180.000} C_DIS
LIN {X 99.221,Y 58.038,Z 62.000,A 180.000,B 0.000,C 180.000} C_DIS
LIN {X 99.395,Y 57.925,Z 62.000,A 180.000,B 0.000,C 180.000} C_DIS
LIN {X 99.757,Y 57.673,Z 62.000,A 180.000,B 0.000,C 180.000} C_DIS
LIN {X 99.909,Y 57.567,Z 62.000,A 180.000,B 0.000,C 180.000} C_DIS
LIN {X 99.936,Y 57.548,Z 62.000,A 180.000,B 0.000,C 180.000} C_DIS
LIN {X 100.114,Y 57.409,Z 62.000,A 180.000,B 0.000,C 180.000} C_DIS
LIN {X 100.472,Y 57.125,Z 62.000,A 180.000,B 0.000,C 180.000} C_DIS
LIN {X 100.588,Y 57.031,Z 62.000,A 180.000,B 0.000,C 180.000} C_DIS
LIN {X 100.651,Y 56.975,Z 62.000,A 180.000,B 0.000,C 180.000} C_DIS
LIN {X 101.008,Y 56.653,Z 62.000,A 180.000,B 0.000,C 180.000} C_DIS
LIN {X 101.180,Y 56.495,Z 62.000,A 180.000,B 0.000,C 180.000} C_DIS
LIN {X 101.187,Y 56.488,Z 62.000,A 180.000,B 0.000,C 180.000} C_DIS
LIN {X 101.356,Y 56.316,Z 62.000,A 180.000,B 0.000,C 180.000} C_DIS
LIN {X 101.545,Y 56.123,Z 62.000,A 180.000,B 0.000,C 180.000} C_DIS
LIN {X 101.704,Y 55.958,Z 62.000,A 180.000,B 0.000,C 180.000} C_DIS
LIN {X 101.723,Y 55.937,Z 62.000,A 180.000,B 0.000,C 180.000} C_DIS
LIN {X 101.860,Y 55.779,Z 62.000,A 180.000,B 0.000,C 180.000} C_DIS
LIN {X 102.168,Y 55.422,Z 62.000,A 180.000,B 0.000,C 180.000} C_DIS
LIN {X 102.260,Y 55.309,Z 62.000,A 180.000,B 0.000,C 180.000} C_DIS
LIN {X 102.310,Y 55.243,Z 62.000,A 180.000,B 0.000,C 180.000} C_DIS
LIN {X 102.617,Y 54.837,Z 62.000,A 180.000,B 0.000,C 180.000} C_DIS
LIN {X 102.713,Y 54.707,Z 62.000,A 180.000,B 0.000,C 180.000} C_DIS
LIN {X 102.796,Y 54.583,Z 62.000,A 180.000,B 0.000,C 180.000} C_DIS
LIN {X 103.069,Y 54.171,Z 62.000,A 180.000,B 0.000,C 180.000} C_DIS
LIN {X 103.153,Y 54.038,Z 62.000,A 180.000,B 0.000,C 180.000} C_DIS
LIN {X 103.180,Y 53.992,Z 62.000,A 180.000,B 0.000,C 180.000} C_DIS
LIN {X 103.386,Y 53.634,Z 62.000,A 180.000,B 0.000,C 180.000} C_DIS
LIN {X 103.489,Y 53.455,Z 62.000,A 180.000,B 0.000,C 180.000} C_DIS
LIN {X 103.511,Y 53.417,Z 62.000,A 180.000,B 0.000,C 180.000} C_DIS
LIN {X 103.583,Y 53.277,Z 62.000,A 180.000,B 0.000,C 180.000} C_DIS
LIN {X 103.760,Y 52.919,Z 62.000,A 180.000,B 0.000,C 180.000} C_DIS
LIN {X 103.848,Y 52.740,Z 62.000,A 180.000,B 0.000,C 180.000} C_DIS
LIN {X 103.869,Y 52.697,Z 62.000,A 180.000,B 0.000,C 180.000} C_DIS
LIN {X 103.927,Y 52.562,Z 62.000,A 180.000,B 0.000,C 180.000} C_DIS
LIN {X 104.077,Y 52.204,Z 62.000,A 180.000,B 0.000,C 180.000} C_DIS
LIN {X 104.152,Y 52.025,Z 62.000,A 180.000,B 0.000,C 180.000} C_DIS
LIN {X 104.218,Y 51.847,Z 62.000,A 180.000,B 0.000,C 180.000} C_DIS
LIN {X 104.405,Y 51.307,Z 62.000,A 180.000,B 0.000,C 180.000} C_DIS
LIN {X 104.459,Y 51.131,Z 62.000,A 180.000,B 0.000,C 180.000} C_DIS
LIN {X 104.609,Y 50.595,Z 62.000,A 180.000,B 0.000,C 180.000} C_DIS
LIN {X 104.654,Y 50.416,Z 62.000,A 180.000,B 0.000,C 180.000} C_DIS
LIN {X 104.692,Y 50.238,Z 62.000,A 180.000,B 0.000,C 180.000} C_DIS
LIN {X 104.768,Y 49.880,Z 62.000,A 180.000,B 0.000,C 180.000} C_DIS
LIN {X 104.805,Y 49.701,Z 62.000,A 180.000,B 0.000,C 180.000} C_DIS
LIN {X 104.832,Y 49.523,Z 62.000,A 180.000,B 0.000,C 180.000} C_DIS
LIN {X 104.885,Y 49.165,Z 62.000,A 180.000,B 0.000,C 180.000} C_DIS
LIN {X 104.911,Y 48.986,Z 62.000,A 180.000,B 0.000,C 180.000} C_DIS
LIN {X 104.929,Y 48.807,Z 62.000,A 180.000,B 0.000,C 180.000} C_DIS
LIN {X 104.974,Y 48.271,Z 62.000,A 180.000,B 0.000,C 180.000} C_DIS
LIN {X 104.986,Y 48.092,Z 62.000,A 180.000,B 0.000,C 180.000} C_DIS
LIN {X 104.989,Y 47.914,Z 62.000,A 180.000,B 0.000,C 180.000} C_DIS
LIN {X 104.996,Y 47.556,Z 62.000,A 180.000,B 0.000,C 180.000} C_DIS
LIN {X 104.999,Y 47.377,Z 62.000,A 180.000,B 0.000,C 180.000} C_DIS
LIN {X 104.994,Y 47.198,Z 62.000,A 180.000,B 0.000,C 180.000} C_DIS
LIN {X 104.971,Y 46.662,Z 62.000,A 180.000,B 0.000,C 180.000} C_DIS
LIN {X 104.957,Y 46.483,Z 62.000,A 180.000,B 0.000,C 180.000} C_DIS
LIN {X 104.900,Y 45.947,Z 62.000,A 180.000,B 0.000,C 180.000} C_DIS
LIN {X 104.879,Y 45.768,Z 62.000,A 180.000,B 0.000,C 180.000} C_DIS
LIN {X 104.850,Y 45.590,Z 62.000,A 180.000,B 0.000,C 180.000} C_DIS
LIN {X 104.789,Y 45.232,Z 62.000,A 180.000,B 0.000,C 180.000} C_DIS
LIN {X 104.762,Y 45.077,Z 62.000,A 180.000,B 0.000,C 180.000} C_DIS
LIN {X 104.758,Y 45.053,Z 62.000,A 180.000,B 0.000,C 180.000} C_DIS
LIN {X 104.719,Y 44.874,Z 62.000,A 180.000,B 0.000,C 180.000} C_DIS
LIN {X 104.592,Y 44.338,Z 62.000,A 180.000,B 0.000,C 180.000} C_DIS
LIN {X 104.584,Y 44.302,Z 62.000,A 180.000,B 0.000,C 180.000} C_DIS
LIN {X 104.544,Y 44.159,Z 62.000,A 180.000,B 0.000,C 180.000} C_DIS
LIN {X 104.381,Y 43.623,Z 62.000,A 180.000,B 0.000,C 180.000} C_DIS
LIN {X 104.323,Y 43.444,Z 62.000,A 180.000,B 0.000,C 180.000} C_DIS
LIN {X 104.257,Y 43.266,Z 62.000,A 180.000,B 0.000,C 180.000} C_DIS
LIN {X 104.123,Y 42.908,Z 62.000,A 180.000,B 0.000,C 180.000} C_DIS
LIN {X 104.053,Y 42.729,Z 62.000,A 180.000,B 0.000,C 180.000} C_DIS
LIN {X 104.047,Y 42.715,Z 62.000,A 180.000,B 0.000,C 180.000} C_DIS
LIN {X 103.974,Y 42.550,Z 62.000,A 180.000,B 0.000,C 180.000} C_DIS
LIN {X 103.814,Y 42.193,Z 62.000,A 180.000,B 0.000,C 180.000} C_DIS
LIN {X 103.732,Y 42.014,Z 62.000,A 180.000,B 0.000,C 180.000} C_DIS
LIN {X 103.690,Y 41.934,Z 62.000,A 180.000,B 0.000,C 180.000} C_DIS
LIN {X 103.451,Y 41.478,Z 62.000,A 180.000,B 0.000,C 180.000} C_DIS
LIN {X 103.353,Y 41.299,Z 62.000,A 180.000,B 0.000,C 180.000} C_DIS
LIN {X 103.332,Y 41.265,Z 62.000,A 180.000,B 0.000,C 180.000} C_DIS
LIN {X 103.027,Y 40.763,Z 62.000,A 180.000,B 0.000,C 180.000} C_DIS
LIN {X 102.975,Y 40.679,Z 62.000,A 180.000,B 0.000,C 180.000} C_DIS
LIN {X 102.910,Y 40.584,Z 62.000,A 180.000,B 0.000,C 180.000} C_DIS
LIN {X 102.617,Y 40.163,Z 62.000,A 180.000,B 0.000,C 180.000} C_DIS
LIN {X 102.536,Y 40.048,Z 62.000,A 180.000,B 0.000,C 180.000} C_DIS
LIN {X 102.438,Y 39.923,Z 62.000,A 180.000,B 0.000,C 180.000} C_DIS
LIN {X 102.112,Y 39.511,Z 62.000,A 180.000,B 0.000,C 180.000} C_DIS
LIN {X 102.081,Y 39.472,Z 62.000,A 180.000,B 0.000,C 180.000} C_DIS
LIN {X 101.960,Y 39.333,Z 62.000,A 180.000,B 0.000,C 180.000} C_DIS
LIN {X 101.638,Y 38.975,Z 62.000,A 180.000,B 0.000,C 180.000} C_DIS
LIN {X 101.545,Y 38.872,Z 62.000,A 180.000,B 0.000,C 180.000} C_DIS
LIN {X 101.471,Y 38.796,Z 62.000,A 180.000,B 0.000,C 180.000} C_DIS
LIN {X 101.366,Y 38.693,Z 62.000,A 180.000,B 0.000,C 180.000} C_DIS
LIN {X 101.008,Y 38.344,Z 62.000,A 180.000,B 0.000,C 180.000} C_DIS
LIN {X 100.918,Y 38.260,Z 62.000,A 180.000,B 0.000,C 180.000} C_DIS
LIN {X 100.829,Y 38.183,Z 62.000,A 180.000,B 0.000,C 180.000} C_DIS
LIN {X 100.472,Y 37.875,Z 62.000,A 180.000,B 0.000,C 180.000} C_DIS
LIN {X 100.293,Y 37.728,Z 62.000,A 180.000,B 0.000,C 180.000} C_DIS
LIN {X 100.003,Y 37.508,Z 62.000,A 180.000,B 0.000,C 180.000} C_DIS
LIN {X 99.815,Y 37.366,Z 62.000,A 180.000,B 0.000,C 180.000} C_DIS
LIN {X 99.757,Y 37.322,Z 62.000,A 180.000,B 0.000,C 180.000} C_DIS
LIN {X 99.578,Y 37.201,Z 62.000,A 180.000,B 0.000,C 180.000} C_DIS
LIN {X 99.221,Y 36.964,Z 62.000,A 180.000,B 0.000,C 180.000} C_DIS
LIN {X 99.042,Y 36.849,Z 62.000,A 180.000,B 0.000,C 180.000} C_DIS
LIN {X 99.009,Y 36.830,Z 62.000,A 180.000,B 0.000,C 180.000} C_DIS
LIN {X 98.505,Y 36.539,Z 62.000,A 180.000,B 0.000,C 180.000} C_DIS
LIN {X 98.385,Y 36.472,Z 62.000,A 180.000,B 0.000,C 180.000} C_DIS
LIN {X 98.327,Y 36.442,Z 62.000,A 180.000,B 0.000,C 180.000} C_DIS
LIN {X 97.790,Y 36.177,Z 62.000,A 180.000,B 0.000,C 180.000} C_DIS
LIN {X 97.659,Y 36.115,Z 62.000,A 180.000,B 0.000,C 180.000} C_DIS
LIN {X 97.612,Y 36.094,Z 62.000,A 180.000,B 0.000,C 180.000} C_DIS
LIN {X 97.075,Y 35.869,Z 62.000,A 180.000,B 0.000,C 180.000} C_DIS
LIN {X 96.897,Y 35.800,Z 62.000,A 180.000,B 0.000,C 180.000} C_DIS
LIN {X 96.360,Y 35.613,Z 62.000,A 180.000,B 0.000,C 180.000} C_DIS
LIN {X 96.258,Y 35.578,Z 62.000,A 180.000,B 0.000,C 180.000} C_DIS
LIN {X 96.181,Y 35.555,Z 62.000,A 180.000,B 0.000,C 180.000} C_DIS
LIN {X 96.003,Y 35.505,Z 62.000,A 180.000,B 0.000,C 180.000} C_DIS
LIN {X 95.625,Y 35.400,Z 62.000,A 180.000,B 0.000,C 180.000} C_DIS
LIN {X 95.466,Y 35.357,Z 62.000,A 180.000,B 0.000,C 180.000} C_DIS
LIN {X 95.288,Y 35.318,Z 62.000,A 180.000,B 0.000,C 180.000} C_DIS
LIN {X 94.828,Y 35.221,Z 62.000,A 180.000,B 0.000,C 180.000} C_DIS
LIN {X 94.751,Y 35.205,Z 62.000,A 180.000,B 0.000,C 180.000} C_DIS
LIN {X 94.573,Y 35.175,Z 62.000,A 180.000,B 0.000,C 180.000} C_DIS
LIN {X 94.036,Y 35.097,Z 62.000,A 180.000,B 0.000,C 180.000} C_DIS
LIN {X 93.857,Y 35.075,Z 62.000,A 180.000,B 0.000,C 180.000} C_DIS
LIN {X 93.679,Y 35.060,Z 62.000,A 180.000,B 0.000,C 180.000} C_DIS
LIN {X 93.321,Y 35.030,Z 62.000,A 180.000,B 0.000,C 180.000} C_DIS
LIN {X 93.142,Y 35.017,Z 62.000,A 180.000,B 0.000,C 180.000} C_DIS
LIN {X 92.964,Y 35.012,Z 62.000,A 180.000,B 0.000,C 180.000} C_DIS
LIN {X 92.606,Y 35.005,Z 62.000,A 180.000,B 0.000,C 180.000} C_DIS
LIN {X 92.427,Y 35.001,Z 62.000,A 180.000,B 0.000,C 180.000} C_DIS
LIN {X 92.249,Y 35.004,Z 62.000,A 180.000,B 0.000,C 180.000} C_DIS
LIN {X 91.712,Y 35.027,Z 62.000,A 180.000,B 0.000,C 180.000} C_DIS
LIN {X 91.533,Y 35.038,Z 62.000,A 180.000,B 0.000,C 180.000} C_DIS
LIN {X 91.489,Y 35.042,Z 62.000,A 180.000,B 0.000,C 180.000} C_DIS
LIN {X 90.997,Y 35.094,Z 62.000,A 180.000,B 0.000,C 180.000} C_DIS
LIN {X 90.818,Y 35.114,Z 62.000,A 180.000,B 0.000,C 180.000} C_DIS
LIN {X 90.640,Y 35.142,Z 62.000,A 180.000,B 0.000,C 180.000} C_DIS
LIN {X 90.103,Y 35.233,Z 62.000,A 180.000,B 0.000,C 180.000} C_DIS
LIN {X 89.925,Y 35.270,Z 62.000,A 180.000,B 0.000,C 180.000} C_DIS
LIN {X 89.372,Y 35.400,Z 62.000,A 180.000,B 0.000,C 180.000} C_DIS
LIN {X 89.209,Y 35.441,Z 62.000,A 180.000,B 0.000,C 180.000} C_DIS
LIN {X 89.031,Y 35.495,Z 62.000,A 180.000,B 0.000,C 180.000} C_DIS
LIN {X 88.673,Y 35.603,Z 62.000,A 180.000,B 0.000,C 180.000} C_DIS
LIN {X 88.494,Y 35.659,Z 62.000,A 180.000,B 0.000,C 180.000} C_DIS
LIN {X 82.417,Y 37.709,Z 62.000,A 180.000,B 0.000,C 180.000} C_DIS
; Lead Out Move Starts
LIN {X 81.963,Y 37.640,Z 62.000,A 180.000,B 0.000,C 180.000} C_DIS
LIN {X 81.757,Y 37.229,Z 62.000,A 180.000,B 0.000,C 180.000} C_DIS
LIN {X 81.770,Y 36.314,Z 62.000,A 180.000,B 0.000,C 180.000} C_DIS
LIN {X 81.775,Y 35.960,Z 62.146,A 180.000,B 0.000,C 180.000} C_DIS
LIN {X 81.777,Y 35.814,Z 62.500,A 180.000,B 0.000,C 180.000} C_DIS
; Rapid Move Starts
LIN {X 81.777,Y 35.814,Z 95.000,A 180.000,B 0.000,C 180.000} C_DIS
LIN {X 77.776,Y 71.334,Z 95.000,A 180.000,B 0.000,C 180.000} C_DIS
LIN {X 77.776,Y 71.334,Z 63.500,A 180.000,B 0.000,C 180.000} C_DIS
; Plunge Move Starts
$VEL.CP=0.01
LIN {X 77.776,Y 71.334,Z 62.625,A 180.000,B 0.000,C 180.000} C_DIS
; Lead In Move Starts
LIN {X 77.776,Y 71.334,Z 61.500,A 180.000,B 0.000,C 180.000} C_DIS
LIN {X 77.799,Y 71.189,Z 61.146,A 180.000,B 0.000,C 180.000} C_DIS
LIN {X 77.855,Y 70.840,Z 61.000,A 180.000,B 0.000,C 180.000} C_DIS
LIN {X 77.911,Y 70.483,Z 61.000,A 180.000,B 0.000,C 180.000} C_DIS
LIN {X 78.111,Y 70.157,Z 61.000,A 180.000,B 0.000,C 180.000} C_DIS
LIN {X 78.483,Y 70.067,Z 61.000,A 180.000,B 0.000,C 180.000} C_DIS
; Cutting Move Starts
$VEL.CP=0.02
LIN {X 78.841,Y 70.124,Z 61.000,A 180.000,B 0.000,C 180.000} C_DIS
LIN {X 79.020,Y 70.160,Z 61.000,A 180.000,B 0.000,C 180.000} C_DIS
LIN {X 79.198,Y 70.200,Z 61.000,A 180.000,B 0.000,C 180.000} C_DIS
LIN {X 79.377,Y 70.240,Z 61.000,A 180.000,B 0.000,C 180.000} C_DIS
LIN {X 79.735,Y 70.344,Z 61.000,A 180.000,B 0.000,C 180.000} C_DIS
LIN {X 79.913,Y 70.403,Z 61.000,A 180.000,B 0.000,C 180.000} C_DIS
LIN {X 80.092,Y 70.467,Z 61.000,A 180.000,B 0.000,C 180.000} C_DIS
LIN {X 80.271,Y 70.532,Z 61.000,A 180.000,B 0.000,C 180.000} C_DIS
LIN {X 80.628,Y 70.687,Z 61.000,A 180.000,B 0.000,C 180.000} C_DIS
LIN {X 80.807,Y 70.773,Z 61.000,A 180.000,B 0.000,C 180.000} C_DIS
LIN {X 80.986,Y 70.864,Z 61.000,A 180.000,B 0.000,C 180.000} C_DIS
LIN {X 81.165,Y 70.960,Z 61.000,A 180.000,B 0.000,C 180.000} C_DIS
LIN {X 81.493,Y 71.154,Z 61.000,A 180.000,B 0.000,C 180.000} C_DIS
LIN {X 81.522,Y 71.171,Z 61.000,A 180.000,B 0.000,C 180.000} C_DIS
LIN {X 81.880,Y 71.414,Z 61.000,A 180.000,B 0.000,C 180.000} C_DIS
LIN {X 82.008,Y 71.511,Z 61.000,A 180.000,B 0.000,C 180.000} C_DIS
LIN {X 82.238,Y 71.690,Z 61.000,A 180.000,B 0.000,C 180.000} C_DIS
LIN {X 82.416,Y 71.842,Z 61.000,A 180.000,B 0.000,C 180.000} C_DIS
LIN {X 82.595,Y 72.000,Z 61.000,A 180.000,B 0.000,C 180.000} C_DIS
LIN {X 82.647,Y 72.048,Z 61.000,A 180.000,B 0.000,C 180.000} C_DIS
LIN {X 82.952,Y 72.353,Z 61.000,A 180.000,B 0.000,C 180.000} C_DIS
LIN {X 83.000,Y 72.405,Z 61.000,A 180.000,B 0.000,C 180.000} C_DIS
LIN {X 83.158,Y 72.584,Z 61.000,A 180.000,B 0.000,C 180.000} C_DIS
LIN {X 83.310,Y 72.762,Z 61.000,A 180.000,B 0.000,C 180.000} C_DIS
LIN {X 83.489,Y 72.992,Z 61.000,A 180.000,B 0.000,C 180.000} C_DIS
LIN {X 83.586,Y 73.120,Z 61.000,A 180.000,B 0.000,C 180.000} C_DIS
LIN {X 83.829,Y 73.478,Z 61.000,A 180.000,B 0.000,C 180.000} C_DIS
LIN {X 83.846,Y 73.507,Z 61.000,A 180.000,B 0.000,C 180.000} C_DIS
LIN {X 84.040,Y 73.835,Z 61.000,A 180.000,B 0.000,C 180.000} C_DIS
LIN {X 84.136,Y 74.014,Z 61.000,A 180.000,B 0.000,C 180.000} C_DIS
LIN {X 84.227,Y 74.193,Z 61.000,A 180.000,B 0.000,C 180.000} C_DIS
LIN {X 84.313,Y 74.372,Z 61.000,A 180.000,B 0.000,C 180.000} C_DIS
LIN {X 84.468,Y 74.729,Z 61.000,A 180.000,B 0.000,C 180.000} C_DIS
LIN {X 84.533,Y 74.908,Z 61.000,A 180.000,B 0.000,C 180.000} C_DIS
LIN {X 84.597,Y 75.087,Z 61.000,A 180.000,B 0.000,C 180.000} C_DIS
LIN {X 84.656,Y 75.265,Z 61.000,A 180.000,B 0.000,C 180.000} C_DIS
LIN {X 84.760,Y 75.623,Z 61.000,A 180.000,B 0.000,C 180.000} C_DIS
LIN {X 84.800,Y 75.802,Z 61.000,A 180.000,B 0.000,C 180.000} C_DIS
LIN {X 84.840,Y 75.980,Z 61.000,A 180.000,B 0.000,C 180.000} C_DIS
LIN {X 84.876,Y 76.159,Z 61.000,A 180.000,B 0.000,C 180.000} C_DIS
LIN {X 84.933,Y 76.517,Z 61.000,A 180.000,B 0.000,C 180.000} C_DIS
LIN {X 84.952,Y 76.696,Z 61.000,A 180.000,B 0.000,C 180.000} C_DIS
LIN {X 84.969,Y 76.874,Z 61.000,A 180.000,B 0.000,C 180.000} C_DIS
LIN {X 84.985,Y 77.053,Z 61.000,A 180.000,B 0.000,C 180.000} C_DIS
LIN {X 84.996,Y 77.411,Z 61.000,A 180.000,B 0.000,C 180.000} C_DIS
LIN {X 84.996,Y 77.589,Z 61.000,A 180.000,B 0.000,C 180.000} C_DIS
LIN {X 84.985,Y 77.947,Z 61.000,A 180.000,B 0.000,C 180.000} C_DIS
LIN {X 84.969,Y 78.126,Z 61.000,A 180.000,B 0.000,C 180.000} C_DIS
LIN {X 84.952,Y 78.304,Z 61.000,A 180.000,B 0.000,C 180.000} C_DIS
LIN {X 84.933,Y 78.483,Z 61.000,A 180.000,B 0.000,C 180.000} C_DIS
LIN {X 84.876,Y 78.841,Z 61.000,A 180.000,B 0.000,C 180.000} C_DIS
LIN {X 84.840,Y 79.020,Z 61.000,A 180.000,B 0.000,C 180.000} C_DIS
LIN {X 84.800,Y 79.198,Z 61.000,A 180.000,B 0.000,C 180.000} C_DIS
LIN {X 84.760,Y 79.377,Z 61.000,A 180.000,B 0.000,C 180.000} C_DIS
LIN {X 84.656,Y 79.735,Z 61.000,A 180.000,B 0.000,C 180.000} C_DIS
LIN {X 84.597,Y 79.913,Z 61.000,A 180.000,B 0.000,C 180.000} C_DIS
LIN {X 84.533,Y 80.092,Z 61.000,A 180.000,B 0.000,C 180.000} C_DIS
LIN {X 84.468,Y 80.271,Z 61.000,A 180.000,B 0.000,C 180.000} C_DIS
LIN {X 84.313,Y 80.628,Z 61.000,A 180.000,B 0.000,C 180.000} C_DIS
LIN {X 84.227,Y 80.807,Z 61.000,A 180.000,B 0.000,C 180.000} C_DIS
LIN {X 84.136,Y 80.986,Z 61.000,A 180.000,B 0.000,C 180.000} C_DIS
LIN {X 84.040,Y 81.165,Z 61.000,A 180.000,B 0.000,C 180.000} C_DIS
LIN {X 83.846,Y 81.493,Z 61.000,A 180.000,B 0.000,C 180.000} C_DIS
LIN {X 83.829,Y 81.522,Z 61.000,A 180.000,B 0.000,C 180.000} C_DIS
LIN {X 83.586,Y 81.880,Z 61.000,A 180.000,B 0.000,C 180.000} C_DIS
LIN {X 83.489,Y 82.008,Z 61.000,A 180.000,B 0.000,C 180.000} C_DIS
LIN {X 83.310,Y 82.238,Z 61.000,A 180.000,B 0.000,C 180.000} C_DIS
LIN {X 83.158,Y 82.416,Z 61.000,A 180.000,B 0.000,C 180.000} C_DIS
LIN {X 83.000,Y 82.595,Z 61.000,A 180.000,B 0.000,C 180.000} C_DIS
LIN {X 82.952,Y 82.647,Z 61.000,A 180.000,B 0.000,C 180.000} C_DIS
LIN {X 82.647,Y 82.952,Z 61.000,A 180.000,B 0.000,C 180.000} C_DIS
LIN {X 82.595,Y 83.000,Z 61.000,A 180.000,B 0.000,C 180.000} C_DIS
LIN {X 82.416,Y 83.158,Z 61.000,A 180.000,B 0.000,C 180.000} C_DIS
LIN {X 82.238,Y 83.310,Z 61.000,A 180.000,B 0.000,C 180.000} C_DIS
LIN {X 82.008,Y 83.489,Z 61.000,A 180.000,B 0.000,C 180.000} C_DIS
LIN {X 81.880,Y 83.586,Z 61.000,A 180.000,B 0.000,C 180.000} C_DIS
LIN {X 81.522,Y 83.829,Z 61.000,A 180.000,B 0.000,C 180.000} C_DIS
LIN {X 81.493,Y 83.846,Z 61.000,A 180.000,B 0.000,C 180.000} C_DIS
LIN {X 81.165,Y 84.040,Z 61.000,A 180.000,B 0.000,C 180.000} C_DIS
LIN {X 80.986,Y 84.136,Z 61.000,A 180.000,B 0.000,C 180.000} C_DIS
LIN {X 80.807,Y 84.227,Z 61.000,A 180.000,B 0.000,C 180.000} C_DIS
LIN {X 80.628,Y 84.313,Z 61.000,A 180.000,B 0.000,C 180.000} C_DIS
LIN {X 80.271,Y 84.468,Z 61.000,A 180.000,B 0.000,C 180.000} C_DIS
LIN {X 80.092,Y 84.533,Z 61.000,A 180.000,B 0.000,C 180.000} C_DIS
LIN {X 79.913,Y 84.597,Z 61.000,A 180.000,B 0.000,C 180.000} C_DIS
LIN {X 79.735,Y 84.656,Z 61.000,A 180.000,B 0.000,C 180.000} C_DIS
LIN {X 79.377,Y 84.760,Z 61.000,A 180.000,B 0.000,C 180.000} C_DIS
LIN {X 79.198,Y 84.800,Z 61.000,A 180.000,B 0.000,C 180.000} C_DIS
LIN {X 79.020,Y 84.840,Z 61.000,A 180.000,B 0.000,C 180.000} C_DIS
LIN {X 78.841,Y 84.876,Z 61.000,A 180.000,B 0.000,C 180.000} C_DIS
LIN {X 78.483,Y 84.933,Z 61.000,A 180.000,B 0.000,C 180.000} C_DIS
LIN {X 78.304,Y 84.952,Z 61.000,A 180.000,B 0.000,C 180.000} C_DIS
LIN {X 78.126,Y 84.969,Z 61.000,A 180.000,B 0.000,C 180.000} C_DIS
LIN {X 77.947,Y 84.985,Z 61.000,A 180.000,B 0.000,C 180.000} C_DIS
LIN {X 77.589,Y 84.996,Z 61.000,A 180.000,B 0.000,C 180.000} C_DIS
LIN {X 77.411,Y 84.996,Z 61.000,A 180.000,B 0.000,C 180.000} C_DIS
LIN {X 77.053,Y 84.985,Z 61.000,A 180.000,B 0.000,C 180.000} C_DIS
LIN {X 76.874,Y 84.969,Z 61.000,A 180.000,B 0.000,C 180.000} C_DIS
LIN {X 76.696,Y 84.952,Z 61.000,A 180.000,B 0.000,C 180.000} C_DIS
LIN {X 76.517,Y 84.933,Z 61.000,A 180.000,B 0.000,C 180.000} C_DIS
LIN {X 76.159,Y 84.876,Z 61.000,A 180.000,B 0.000,C 180.000} C_DIS
LIN {X 75.980,Y 84.840,Z 61.000,A 180.000,B 0.000,C 180.000} C_DIS
LIN {X 75.802,Y 84.800,Z 61.000,A 180.000,B 0.000,C 180.000} C_DIS
LIN {X 75.623,Y 84.760,Z 61.000,A 180.000,B 0.000,C 180.000} C_DIS
LIN {X 75.265,Y 84.656,Z 61.000,A 180.000,B 0.000,C 180.000} C_DIS
LIN {X 75.087,Y 84.597,Z 61.000,A 180.000,B 0.000,C 180.000} C_DIS
LIN {X 74.908,Y 84.533,Z 61.000,A 180.000,B 0.000,C 180.000} C_DIS
LIN {X 74.729,Y 84.468,Z 61.000,A 180.000,B 0.000,C 180.000} C_DIS
LIN {X 74.372,Y 84.313,Z 61.000,A 180.000,B 0.000,C 180.000} C_DIS
LIN {X 74.193,Y 84.227,Z 61.000,A 180.000,B 0.000,C 180.000} C_DIS
LIN {X 74.014,Y 84.136,Z 61.000,A 180.000,B 0.000,C 180.000} C_DIS
LIN {X 73.835,Y 84.040,Z 61.000,A 180.000,B 0.000,C 180.000} C_DIS
LIN {X 73.507,Y 83.846,Z 61.000,A 180.000,B 0.000,C 180.000} C_DIS
LIN {X 73.478,Y 83.829,Z 61.000,A 180.000,B 0.000,C 180.000} C_DIS
LIN {X 73.120,Y 83.586,Z 61.000,A 180.000,B 0.000,C 180.000} C_DIS
LIN {X 72.992,Y 83.489,Z 61.000,A 180.000,B 0.000,C 180.000} C_DIS
LIN {X 72.762,Y 83.310,Z 61.000,A 180.000,B 0.000,C 180.000} C_DIS
LIN {X 72.584,Y 83.158,Z 61.000,A 180.000,B 0.000,C 180.000} C_DIS
LIN {X 72.405,Y 83.000,Z 61.000,A 180.000,B 0.000,C 180.000} C_DIS
LIN {X 72.353,Y 82.952,Z 61.000,A 180.000,B 0.000,C 180.000} C_DIS
LIN {X 72.048,Y 82.647,Z 61.000,A 180.000,B 0.000,C 180.000} C_DIS
LIN {X 72.000,Y 82.595,Z 61.000,A 180.000,B 0.000,C 180.000} C_DIS
LIN {X 71.842,Y 82.416,Z 61.000,A 180.000,B 0.000,C 180.000} C_DIS
LIN {X 71.690,Y 82.238,Z 61.000,A 180.000,B 0.000,C 180.000} C_DIS
LIN {X 71.511,Y 82.008,Z 61.000,A 180.000,B 0.000,C 180.000} C_DIS
LIN {X 71.414,Y 81.880,Z 61.000,A 180.000,B 0.000,C 180.000} C_DIS
LIN {X 71.171,Y 81.522,Z 61.000,A 180.000,B 0.000,C 180.000} C_DIS
LIN {X 71.154,Y 81.493,Z 61.000,A 180.000,B 0.000,C 180.000} C_DIS
LIN {X 70.960,Y 81.165,Z 61.000,A 180.000,B 0.000,C 180.000} C_DIS
LIN {X 70.864,Y 80.986,Z 61.000,A 180.000,B 0.000,C 180.000} C_DIS
LIN {X 70.773,Y 80.807,Z 61.000,A 180.000,B 0.000,C 180.000} C_DIS
LIN {X 70.687,Y 80.628,Z 61.000,A 180.000,B 0.000,C 180.000} C_DIS
LIN {X 70.532,Y 80.271,Z 61.000,A 180.000,B 0.000,C 180.000} C_DIS
LIN {X 70.467,Y 80.092,Z 61.000,A 180.000,B 0.000,C 180.000} C_DIS
LIN {X 70.403,Y 79.913,Z 61.000,A 180.000,B 0.000,C 180.000} C_DIS
LIN {X 70.344,Y 79.735,Z 61.000,A 180.000,B 0.000,C 180.000} C_DIS
LIN {X 70.240,Y 79.377,Z 61.000,A 180.000,B 0.000,C 180.000} C_DIS
LIN {X 70.200,Y 79.198,Z 61.000,A 180.000,B 0.000,C 180.000} C_DIS
LIN {X 70.160,Y 79.020,Z 61.000,A 180.000,B 0.000,C 180.000} C_DIS
LIN {X 70.124,Y 78.841,Z 61.000,A 180.000,B 0.000,C 180.000} C_DIS
LIN {X 70.067,Y 78.483,Z 61.000,A 180.000,B 0.000,C 180.000} C_DIS
LIN {X 70.048,Y 78.304,Z 61.000,A 180.000,B 0.000,C 180.000} C_DIS
LIN {X 70.031,Y 78.126,Z 61.000,A 180.000,B 0.000,C 180.000} C_DIS
LIN {X 70.015,Y 77.947,Z 61.000,A 180.000,B 0.000,C 180.000} C_DIS
LIN {X 70.004,Y 77.589,Z 61.000,A 180.000,B 0.000,C 180.000} C_DIS
LIN {X 70.004,Y 77.411,Z 61.000,A 180.000,B 0.000,C 180.000} C_DIS
LIN {X 70.015,Y 77.053,Z 61.000,A 180.000,B 0.000,C 180.000} C_DIS
LIN {X 70.031,Y 76.874,Z 61.000,A 180.000,B 0.000,C 180.000} C_DIS
LIN {X 70.048,Y 76.696,Z 61.000,A 180.000,B 0.000,C 180.000} C_DIS
LIN {X 70.067,Y 76.517,Z 61.000,A 180.000,B 0.000,C 180.000} C_DIS
LIN {X 70.124,Y 76.159,Z 61.000,A 180.000,B 0.000,C 180.000} C_DIS
LIN {X 70.160,Y 75.980,Z 61.000,A 180.000,B 0.000,C 180.000} C_DIS
LIN {X 70.200,Y 75.802,Z 61.000,A 180.000,B 0.000,C 180.000} C_DIS
LIN {X 70.240,Y 75.623,Z 61.000,A 180.000,B 0.000,C 180.000} C_DIS
LIN {X 70.344,Y 75.265,Z 61.000,A 180.000,B 0.000,C 180.000} C_DIS
LIN {X 70.403,Y 75.087,Z 61.000,A 180.000,B 0.000,C 180.000} C_DIS
LIN {X 70.467,Y 74.908,Z 61.000,A 180.000,B 0.000,C 180.000} C_DIS
LIN {X 70.532,Y 74.729,Z 61.000,A 180.000,B 0.000,C 180.000} C_DIS
LIN {X 70.687,Y 74.372,Z 61.000,A 180.000,B 0.000,C 180.000} C_DIS
LIN {X 70.773,Y 74.193,Z 61.000,A 180.000,B 0.000,C 180.000} C_DIS
LIN {X 70.864,Y 74.014,Z 61.000,A 180.000,B 0.000,C 180.000} C_DIS
LIN {X 70.960,Y 73.835,Z 61.000,A 180.000,B 0.000,C 180.000} C_DIS
LIN {X 71.154,Y 73.507,Z 61.000,A 180.000,B 0.000,C 180.000} C_DIS
LIN {X 71.171,Y 73.478,Z 61.000,A 180.000,B 0.000,C 180.000} C_DIS
LIN {X 71.414,Y 73.120,Z 61.000,A 180.000,B 0.000,C 180.000} C_DIS
LIN {X 71.511,Y 72.992,Z 61.000,A 180.000,B 0.000,C 180.000} C_DIS
LIN {X 71.690,Y 72.762,Z 61.000,A 180.000,B 0.000,C 180.000} C_DIS
LIN {X 71.842,Y 72.584,Z 61.000,A 180.000,B 0.000,C 180.000} C_DIS
LIN {X 72.000,Y 72.405,Z 61.000,A 180.000,B 0.000,C 180.000} C_DIS
LIN {X 72.048,Y 72.353,Z 61.000,A 180.000,B 0.000,C 180.000} C_DIS
LIN {X 72.353,Y 72.048,Z 61.000,A 180.000,B 0.000,C 180.000} C_DIS
LIN {X 72.405,Y 72.000,Z 61.000,A 180.000,B 0.000,C 180.000} C_DIS
LIN {X 72.584,Y 71.842,Z 61.000,A 180.000,B 0.000,C 180.000} C_DIS
LIN {X 72.762,Y 71.690,Z 61.000,A 180.000,B 0.000,C 180.000} C_DIS
LIN {X 72.992,Y 71.511,Z 61.000,A 180.000,B 0.000,C 180.000} C_DIS
LIN {X 73.120,Y 71.414,Z 61.000,A 180.000,B 0.000,C 180.000} C_DIS
LIN {X 73.478,Y 71.171,Z 61.000,A 180.000,B 0.000,C 180.000} C_DIS
LIN {X 73.507,Y 71.154,Z 61.000,A 180.000,B 0.000,C 180.000} C_DIS
LIN {X 73.835,Y 70.960,Z 61.000,A 180.000,B 0.000,C 180.000} C_DIS
LIN {X 74.014,Y 70.864,Z 61.000,A 180.000,B 0.000,C 180.000} C_DIS
LIN {X 74.193,Y 70.773,Z 61.000,A 180.000,B 0.000,C 180.000} C_DIS
LIN {X 74.372,Y 70.687,Z 61.000,A 180.000,B 0.000,C 180.000} C_DIS
LIN {X 74.729,Y 70.532,Z 61.000,A 180.000,B 0.000,C 180.000} C_DIS
LIN {X 74.908,Y 70.467,Z 61.000,A 180.000,B 0.000,C 180.000} C_DIS
LIN {X 75.087,Y 70.403,Z 61.000,A 180.000,B 0.000,C 180.000} C_DIS
LIN {X 75.265,Y 70.344,Z 61.000,A 180.000,B 0.000,C 180.000} C_DIS
LIN {X 75.623,Y 70.240,Z 61.000,A 180.000,B 0.000,C 180.000} C_DIS
LIN {X 75.802,Y 70.200,Z 61.000,A 180.000,B 0.000,C 180.000} C_DIS
LIN {X 75.980,Y 70.160,Z 61.000,A 180.000,B 0.000,C 180.000} C_DIS
LIN {X 76.159,Y 70.124,Z 61.000,A 180.000,B 0.000,C 180.000} C_DIS
LIN {X 76.517,Y 70.067,Z 61.000,A 180.000,B 0.000,C 180.000} C_DIS
LIN {X 76.696,Y 70.048,Z 61.000,A 180.000,B 0.000,C 180.000} C_DIS
LIN {X 76.874,Y 70.031,Z 61.000,A 180.000,B 0.000,C 180.000} C_DIS
LIN {X 77.053,Y 70.015,Z 61.000,A 180.000,B 0.000,C 180.000} C_DIS
LIN {X 77.411,Y 70.004,Z 61.000,A 180.000,B 0.000,C 180.000} C_DIS
LIN {X 77.589,Y 70.004,Z 61.000,A 180.000,B 0.000,C 180.000} C_DIS
LIN {X 77.947,Y 70.015,Z 61.000,A 180.000,B 0.000,C 180.000} C_DIS
LIN {X 78.126,Y 70.031,Z 61.000,A 180.000,B 0.000,C 180.000} C_DIS
LIN {X 78.304,Y 70.048,Z 61.000,A 180.000,B 0.000,C 180.000} C_DIS
LIN {X 78.483,Y 70.067,Z 61.000,A 180.000,B 0.000,C 180.000} C_DIS
; Link Move Starts
LIN {X 78.794,Y 70.117,Z 61.000,A 180.000,B 0.000,C 180.000} C_DIS
LIN {X 79.103,Y 70.178,Z 60.999,A 180.000,B 0.000,C 180.000} C_DIS
LIN {X 79.410,Y 70.250,Z 60.998,A 180.000,B 0.000,C 180.000} C_DIS
LIN {X 79.712,Y 70.338,Z 60.996,A 180.000,B 0.000,C 180.000} C_DIS
LIN {X 80.011,Y 70.438,Z 60.994,A 180.000,B 0.000,C 180.000} C_DIS
LIN {X 80.306,Y 70.548,Z 60.991,A 180.000,B 0.000,C 180.000} C_DIS
LIN {X 80.595,Y 70.673,Z 60.988,A 180.000,B 0.000,C 180.000} C_DIS
LIN {X 80.879,Y 70.810,Z 60.985,A 180.000,B 0.000,C 180.000} C_DIS
LIN {X 81.158,Y 70.956,Z 60.981,A 180.000,B 0.000,C 180.000} C_DIS
LIN {X 81.429,Y 71.116,Z 60.977,A 180.000,B 0.000,C 180.000} C_DIS
LIN {X 81.693,Y 71.288,Z 60.972,A 180.000,B 0.000,C 180.000} C_DIS
LIN {X 81.823,Y 71.376,Z 60.969,A 180.000,B 0.000,C 180.000} C_DIS
LIN {X 81.952,Y 71.468,Z 60.967,A 180.000,B 0.000,C 180.000} C_DIS
LIN {X 82.076,Y 71.564,Z 60.964,A 180.000,B 0.000,C 180.000} C_DIS
LIN {X 82.201,Y 71.661,Z 60.961,A 180.000,B 0.000,C 180.000} C_DIS
LIN {X 82.323,Y 71.760,Z 60.959,A 180.000,B 0.000,C 180.000} C_DIS
LIN {X 82.441,Y 71.864,Z 60.956,A 180.000,B 0.000,C 180.000} C_DIS
LIN {X 82.559,Y 71.968,Z 60.952,A 180.000,B 0.000,C 180.000} C_DIS
LIN {X 82.675,Y 72.075,Z 60.949,A 180.000,B 0.000,C 180.000} C_DIS
LIN {X 82.786,Y 72.186,Z 60.946,A 180.000,B 0.000,C 180.000} C_DIS
LIN {X 82.897,Y 72.298,Z 60.943,A 180.000,B 0.000,C 180.000} C_DIS
LIN {X 83.006,Y 72.412,Z 60.939,A 180.000,B 0.000,C 180.000} C_DIS
LIN {X 83.110,Y 72.530,Z 60.936,A 180.000,B 0.000,C 180.000} C_DIS
LIN {X 83.214,Y 72.648,Z 60.932,A 180.000,B 0.000,C 180.000} C_DIS
LIN {X 83.316,Y 72.769,Z 60.928,A 180.000,B 0.000,C 180.000} C_DIS
LIN {X 83.412,Y 72.893,Z 60.925,A 180.000,B 0.000,C 180.000} C_DIS
LIN {X 83.509,Y 73.018,Z 60.921,A 180.000,B 0.000,C 180.000} C_DIS
LIN {X 83.602,Y 73.144,Z 60.917,A 180.000,B 0.000,C 180.000} C_DIS
LIN {X 83.691,Y 73.275,Z 60.913,A 180.000,B 0.000,C 180.000} C_DIS
LIN {X 83.779,Y 73.405,Z 60.909,A 180.000,B 0.000,C 180.000} C_DIS
LIN {X 83.864,Y 73.537,Z 60.905,A 180.000,B 0.000,C 180.000} C_DIS
LIN {X 83.944,Y 73.673,Z 60.900,A 180.000,B 0.000,C 180.000} C_DIS
LIN {X 84.025,Y 73.809,Z 60.896,A 180.000,B 0.000,C 180.000} C_DIS
LIN {X 84.101,Y 73.946,Z 60.892,A 180.000,B 0.000,C 180.000} C_DIS
LIN {X 84.173,Y 74.087,Z 60.887,A 180.000,B 0.000,C 180.000} C_DIS
LIN {X 84.244,Y 74.227,Z 60.883,A 180.000,B 0.000,C 180.000} C_DIS
LIN {X 84.312,Y 74.369,Z 60.878,A 180.000,B 0.000,C 180.000} C_DIS
LIN {X 84.374,Y 74.514,Z 60.873,A 180.000,B 0.000,C 180.000} C_DIS
LIN {X 84.437,Y 74.658,Z 60.869,A 180.000,B 0.000,C 180.000} C_DIS
LIN {X 84.496,Y 74.804,Z 60.864,A 180.000,B 0.000,C 180.000} C_DIS
LIN {X 84.549,Y 74.953,Z 60.859,A 180.000,B 0.000,C 180.000} C_DIS
LIN {X 84.602,Y 75.101,Z 60.854,A 180.000,B 0.000,C 180.000} C_DIS
LIN {X 84.629,Y 75.175,Z 60.851,A 180.000,B 0.000,C 180.000} C_DIS
LIN {X 84.651,Y 75.250,Z 60.849,A 180.000,B 0.000,C 180.000} C_DIS
LIN {X 84.673,Y 75.326,Z 60.846,A 180.000,B 0.000,C 180.000} C_DIS
LIN {X 84.695,Y 75.402,Z 60.844,A 180.000,B 0.000,C 180.000} C_DIS
LIN {X 84.717,Y 75.477,Z 60.841,A 180.000,B 0.000,C 180.000} C_DIS
LIN {X 84.761,Y 75.628,Z 60.836,A 180.000,B 0.000,C 180.000} C_DIS
LIN {X 84.779,Y 75.705,Z 60.833,A 180.000,B 0.000,C 180.000} C_DIS
LIN {X 84.813,Y 75.859,Z 60.828,A 180.000,B 0.000,C 180.000} C_DIS
LIN {X 84.848,Y 76.013,Z 60.823,A 180.000,B 0.000,C 180.000} C_DIS
LIN {X 84.865,Y 76.090,Z 60.820,A 180.000,B 0.000,C 180.000} C_DIS
LIN {X 84.877,Y 76.167,Z 60.817,A 180.000,B 0.000,C 180.000} C_DIS
LIN {X 84.902,Y 76.323,Z 60.812,A 180.000,B 0.000,C 180.000} C_DIS
LIN {X 84.939,Y 76.556,Z 60.804,A 180.000,B 0.000,C 180.000} C_DIS
LIN {X 84.947,Y 76.635,Z 60.801,A 180.000,B 0.000,C 180.000} C_DIS
LIN {X 84.969,Y 76.870,Z 60.793,A 180.000,B 0.000,C 180.000} C_DIS
LIN {X 84.984,Y 77.027,Z 60.787,A 180.000,B 0.000,C 180.000} C_DIS
LIN {X 84.986,Y 77.105,Z 60.785,A 180.000,B 0.000,C 180.000} C_DIS
LIN {X 84.991,Y 77.263,Z 60.779,A 180.000,B 0.000,C 180.000} C_DIS
LIN {X 84.999,Y 77.499,Z 60.771,A 180.000,B 0.000,C 180.000} C_DIS
LIN {X 84.996,Y 77.578,Z 60.768,A 180.000,B 0.000,C 180.000} C_DIS
LIN {X 84.989,Y 77.814,Z 60.760,A 180.000,B 0.000,C 180.000} C_DIS
LIN {X 84.986,Y 77.893,Z 60.757,A 180.000,B 0.000,C 180.000} C_DIS
LIN {X 84.984,Y 77.971,Z 60.754,A 180.000,B 0.000,C 180.000} C_DIS
LIN {X 84.977,Y 78.050,Z 60.752,A 180.000,B 0.000,C 180.000} C_DIS
LIN {X 84.962,Y 78.207,Z 60.746,A 180.000,B 0.000,C 180.000} C_DIS
LIN {X 84.947,Y 78.363,Z 60.741,A 180.000,B 0.000,C 180.000} C_DIS
LIN {X 84.939,Y 78.442,Z 60.738,A 180.000,B 0.000,C 180.000} C_DIS
LIN {X 84.915,Y 78.597,Z 60.732,A 180.000,B 0.000,C 180.000} C_DIS
LIN {X 84.902,Y 78.675,Z 60.730,A 180.000,B 0.000,C 180.000} C_DIS
LIN {X 84.878,Y 78.831,Z 60.724,A 180.000,B 0.000,C 180.000} C_DIS
LIN {X 84.865,Y 78.908,Z 60.721,A 180.000,B 0.000,C 180.000} C_DIS
LIN {X 84.848,Y 78.985,Z 60.719,A 180.000,B 0.000,C 180.000} C_DIS
LIN {X 84.814,Y 79.139,Z 60.713,A 180.000,B 0.000,C 180.000} C_DIS
LIN {X 84.779,Y 79.293,Z 60.708,A 180.000,B 0.000,C 180.000} C_DIS
LIN {X 84.762,Y 79.370,Z 60.705,A 180.000,B 0.000,C 180.000} C_DIS
LIN {X 84.718,Y 79.521,Z 60.699,A 180.000,B 0.000,C 180.000} C_DIS
LIN {X 84.696,Y 79.596,Z 60.697,A 180.000,B 0.000,C 180.000} C_DIS
LIN {X 84.652,Y 79.748,Z 60.691,A 180.000,B 0.000,C 180.000} C_DIS
LIN {X 84.630,Y 79.823,Z 60.688,A 180.000,B 0.000,C 180.000} C_DIS
LIN {X 84.603,Y 79.897,Z 60.686,A 180.000,B 0.000,C 180.000} C_DIS
LIN {X 84.550,Y 80.046,Z 60.680,A 180.000,B 0.000,C 180.000} C_DIS
LIN {X 84.496,Y 80.194,Z 60.675,A 180.000,B 0.000,C 180.000} C_DIS
LIN {X 84.469,Y 80.268,Z 60.672,A 180.000,B 0.000,C 180.000} C_DIS
LIN {X 84.407,Y 80.412,Z 60.666,A 180.000,B 0.000,C 180.000} C_DIS
LIN {X 84.344,Y 80.557,Z 60.661,A 180.000,B 0.000,C 180.000} C_DIS
LIN {X 84.313,Y 80.629,Z 60.658,A 180.000,B 0.000,C 180.000} C_DIS
LIN {X 84.281,Y 80.701,Z 60.655,A 180.000,B 0.000,C 180.000} C_DIS
LIN {X 84.209,Y 80.841,Z 60.650,A 180.000,B 0.000,C 180.000} C_DIS
LIN {X 84.102,Y 81.052,Z 60.642,A 180.000,B 0.000,C 180.000} C_DIS
LIN {X 84.066,Y 81.122,Z 60.639,A 180.000,B 0.000,C 180.000} C_DIS
LIN {X 83.865,Y 81.461,Z 60.625,A 180.000,B 0.000,C 180.000} C_DIS
LIN {X 83.825,Y 81.528,Z 60.622,A 180.000,B 0.000,C 180.000} C_DIS
LIN {X 83.692,Y 81.724,Z 60.614,A 180.000,B 0.000,C 180.000} C_DIS
LIN {X 83.603,Y 81.854,Z 60.609,A 180.000,B 0.000,C 180.000} C_DIS
LIN {X 83.558,Y 81.919,Z 60.606,A 180.000,B 0.000,C 180.000} C_DIS
LIN {X 83.317,Y 82.230,Z 60.592,A 180.000,B 0.000,C 180.000} C_DIS
LIN {X 83.268,Y 82.291,Z 60.589,A 180.000,B 0.000,C 180.000} C_DIS
LIN {X 83.007,Y 82.587,Z 60.576,A 180.000,B 0.000,C 180.000} C_DIS
LIN {X 82.955,Y 82.645,Z 60.573,A 180.000,B 0.000,C 180.000} C_DIS
LIN {X 82.676,Y 82.923,Z 60.559,A 180.000,B 0.000,C 180.000} C_DIS
LIN {X 82.620,Y 82.978,Z 60.556,A 180.000,B 0.000,C 180.000} C_DIS
LIN {X 82.324,Y 83.239,Z 60.543,A 180.000,B 0.000,C 180.000} C_DIS
LIN {X 82.264,Y 83.290,Z 60.540,A 180.000,B 0.000,C 180.000} C_DIS
LIN {X 81.953,Y 83.531,Z 60.526,A 180.000,B 0.000,C 180.000} C_DIS
LIN {X 81.890,Y 83.578,Z 60.523,A 180.000,B 0.000,C 180.000} C_DIS
LIN {X 81.565,Y 83.800,Z 60.510,A 180.000,B 0.000,C 180.000} C_DIS
LIN {X 81.499,Y 83.843,Z 60.507,A 180.000,B 0.000,C 180.000} C_DIS
LIN {X 81.160,Y 84.043,Z 60.493,A 180.000,B 0.000,C 180.000} C_DIS
LIN {X 81.091,Y 84.082,Z 60.490,A 180.000,B 0.000,C 180.000} C_DIS
LIN {X 80.740,Y 84.261,Z 60.477,A 180.000,B 0.000,C 180.000} C_DIS
LIN {X 80.669,Y 84.295,Z 60.474,A 180.000,B 0.000,C 180.000} C_DIS
LIN {X 80.308,Y 84.452,Z 60.460,A 180.000,B 0.000,C 180.000} C_DIS
LIN {X 80.235,Y 84.481,Z 60.457,A 180.000,B 0.000,C 180.000} C_DIS
LIN {X 79.865,Y 84.615,Z 60.444,A 180.000,B 0.000,C 180.000} C_DIS
LIN {X 79.790,Y 84.640,Z 60.441,A 180.000,B 0.000,C 180.000} C_DIS
LIN {X 79.412,Y 84.750,Z 60.427,A 180.000,B 0.000,C 180.000} C_DIS
LIN {X 79.336,Y 84.770,Z 60.424,A 180.000,B 0.000,C 180.000} C_DIS
LIN {X 79.105,Y 84.821,Z 60.416,A 180.000,B 0.000,C 180.000} C_DIS
LIN {X 78.951,Y 84.856,Z 60.411,A 180.000,B 0.000,C 180.000} C_DIS
LIN {X 78.874,Y 84.871,Z 60.408,A 180.000,B 0.000,C 180.000} C_DIS
LIN {X 78.485,Y 84.932,Z 60.394,A 180.000,B 0.000,C 180.000} C_DIS
LIN {X 78.407,Y 84.943,Z 60.391,A 180.000,B 0.000,C 180.000} C_DIS
LIN {X 78.250,Y 84.958,Z 60.386,A 180.000,B 0.000,C 180.000} C_DIS
LIN {X 78.015,Y 84.980,Z 60.378,A 180.000,B 0.000,C 180.000} C_DIS
LIN {X 77.937,Y 84.985,Z 60.375,A 180.000,B 0.000,C 180.000} C_DIS
LIN {X 77.543,Y 84.997,Z 60.361,A 180.000,B 0.000,C 180.000} C_DIS
LIN {X 77.464,Y 84.998,Z 60.358,A 180.000,B 0.000,C 180.000} C_DIS
LIN {X 77.307,Y 84.993,Z 60.353,A 180.000,B 0.000,C 180.000} C_DIS
LIN {X 77.071,Y 84.985,Z 60.345,A 180.000,B 0.000,C 180.000} C_DIS
LIN {X 76.992,Y 84.980,Z 60.342,A 180.000,B 0.000,C 180.000} C_DIS
LIN {X 76.600,Y 84.943,Z 60.328,A 180.000,B 0.000,C 180.000} C_DIS
LIN {X 76.522,Y 84.934,Z 60.325,A 180.000,B 0.000,C 180.000} C_DIS
LIN {X 76.444,Y 84.921,Z 60.323,A 180.000,B 0.000,C 180.000} C_DIS
LIN {X 76.289,Y 84.897,Z 60.317,A 180.000,B 0.000,C 180.000} C_DIS
LIN {X 76.133,Y 84.872,Z 60.312,A 180.000,B 0.000,C 180.000} C_DIS
LIN {X 76.056,Y 84.857,Z 60.309,A 180.000,B 0.000,C 180.000} C_DIS
LIN {X 75.902,Y 84.823,Z 60.303,A 180.000,B 0.000,C 180.000} C_DIS
LIN {X 75.825,Y 84.806,Z 60.301,A 180.000,B 0.000,C 180.000} C_DIS
LIN {X 75.671,Y 84.771,Z 60.295,A 180.000,B 0.000,C 180.000} C_DIS
LIN {X 75.595,Y 84.752,Z 60.292,A 180.000,B 0.000,C 180.000} C_DIS
LIN {X 75.519,Y 84.730,Z 60.290,A 180.000,B 0.000,C 180.000} C_DIS
LIN {X 75.368,Y 84.686,Z 60.284,A 180.000,B 0.000,C 180.000} C_DIS
LIN {X 75.217,Y 84.642,Z 60.279,A 180.000,B 0.000,C 180.000} C_DIS
LIN {X 75.142,Y 84.617,Z 60.276,A 180.000,B 0.000,C 180.000} C_DIS
LIN {X 74.994,Y 84.564,Z 60.270,A 180.000,B 0.000,C 180.000} C_DIS
LIN {X 74.920,Y 84.537,Z 60.268,A 180.000,B 0.000,C 180.000} C_DIS
LIN {X 74.772,Y 84.484,Z 60.262,A 180.000,B 0.000,C 180.000} C_DIS
LIN {X 74.699,Y 84.454,Z 60.259,A 180.000,B 0.000,C 180.000} C_DIS
LIN {X 74.626,Y 84.423,Z 60.257,A 180.000,B 0.000,C 180.000} C_DIS
LIN {X 74.482,Y 84.361,Z 60.251,A 180.000,B 0.000,C 180.000} C_DIS
LIN {X 74.337,Y 84.298,Z 60.246,A 180.000,B 0.000,C 180.000} C_DIS
LIN {X 74.266,Y 84.264,Z 60.243,A 180.000,B 0.000,C 180.000} C_DIS
LIN {X 74.126,Y 84.193,Z 60.237,A 180.000,B 0.000,C 180.000} C_DIS
LIN {X 74.056,Y 84.157,Z 60.235,A 180.000,B 0.000,C 180.000} C_DIS
LIN {X 73.915,Y 84.085,Z 60.229,A 180.000,B 0.000,C 180.000} C_DIS
LIN {X 73.846,Y 84.047,Z 60.226,A 180.000,B 0.000,C 180.000} C_DIS
LIN {X 73.779,Y 84.007,Z 60.224,A 180.000,B 0.000,C 180.000} C_DIS
LIN {X 73.643,Y 83.927,Z 60.218,A 180.000,B 0.000,C 180.000} C_DIS
LIN {X 73.508,Y 83.847,Z 60.213,A 180.000,B 0.000,C 180.000} C_DIS
LIN {X 73.441,Y 83.804,Z 60.210,A 180.000,B 0.000,C 180.000} C_DIS
LIN {X 73.311,Y 83.715,Z 60.204,A 180.000,B 0.000,C 180.000} C_DIS
LIN {X 73.246,Y 83.671,Z 60.202,A 180.000,B 0.000,C 180.000} C_DIS
LIN {X 73.116,Y 83.583,Z 60.196,A 180.000,B 0.000,C 180.000} C_DIS
LIN {X 73.052,Y 83.536,Z 60.193,A 180.000,B 0.000,C 180.000} C_DIS
LIN {X 72.804,Y 83.343,Z 60.182,A 180.000,B 0.000,C 180.000} C_DIS
LIN {X 72.741,Y 83.294,Z 60.180,A 180.000,B 0.000,C 180.000} C_DIS
LIN {X 72.681,Y 83.244,Z 60.177,A 180.000,B 0.000,C 180.000} C_DIS
LIN {X 72.563,Y 83.139,Z 60.172,A 180.000,B 0.000,C 180.000} C_DIS
LIN {X 72.445,Y 83.035,Z 60.166,A 180.000,B 0.000,C 180.000} C_DIS
LIN {X 72.386,Y 82.983,Z 60.164,A 180.000,B 0.000,C 180.000} C_DIS
LIN {X 72.329,Y 82.929,Z 60.161,A 180.000,B 0.000,C 180.000} C_DIS
LIN {X 72.273,Y 82.873,Z 60.159,A 180.000,B 0.000,C 180.000} C_DIS
LIN {X 72.218,Y 82.817,Z 60.156,A 180.000,B 0.000,C 180.000} C_DIS
LIN {X 72.162,Y 82.762,Z 60.154,A 180.000,B 0.000,C 180.000} C_DIS
LIN {X 72.106,Y 82.706,Z 60.151,A 180.000,B 0.000,C 180.000} C_DIS
LIN {X 72.051,Y 82.650,Z 60.149,A 180.000,B 0.000,C 180.000} C_DIS
LIN {X 71.945,Y 82.533,Z 60.144,A 180.000,B 0.000,C 180.000} C_DIS
LIN {X 71.841,Y 82.415,Z 60.139,A 180.000,B 0.000,C 180.000} C_DIS
LIN {X 71.737,Y 82.297,Z 60.134,A 180.000,B 0.000,C 180.000} C_DIS
LIN {X 71.639,Y 82.173,Z 60.129,A 180.000,B 0.000,C 180.000} C_DIS
LIN {X 71.543,Y 82.049,Z 60.124,A 180.000,B 0.000,C 180.000} C_DIS
LIN {X 71.446,Y 81.924,Z 60.120,A 180.000,B 0.000,C 180.000} C_DIS
LIN {X 71.357,Y 81.795,Z 60.115,A 180.000,B 0.000,C 180.000} C_DIS
LIN {X 71.268,Y 81.664,Z 60.111,A 180.000,B 0.000,C 180.000} C_DIS
LIN {X 71.180,Y 81.534,Z 60.106,A 180.000,B 0.000,C 180.000} C_DIS
LIN {X 71.098,Y 81.399,Z 60.102,A 180.000,B 0.000,C 180.000} C_DIS
LIN {X 71.018,Y 81.264,Z 60.097,A 180.000,B 0.000,C 180.000} C_DIS
LIN {X 70.938,Y 81.128,Z 60.093,A 180.000,B 0.000,C 180.000} C_DIS
LIN {X 70.865,Y 80.988,Z 60.089,A 180.000,B 0.000,C 180.000} C_DIS
LIN {X 70.794,Y 80.848,Z 60.085,A 180.000,B 0.000,C 180.000} C_DIS
LIN {X 70.722,Y 80.708,Z 60.081,A 180.000,B 0.000,C 180.000} C_DIS
LIN {X 70.659,Y 80.563,Z 60.077,A 180.000,B 0.000,C 180.000} C_DIS
LIN {X 70.596,Y 80.419,Z 60.073,A 180.000,B 0.000,C 180.000} C_DIS
LIN {X 70.534,Y 80.274,Z 60.070,A 180.000,B 0.000,C 180.000} C_DIS
LIN {X 70.480,Y 80.126,Z 60.066,A 180.000,B 0.000,C 180.000} C_DIS
LIN {X 70.426,Y 79.978,Z 60.062,A 180.000,B 0.000,C 180.000} C_DIS
LIN {X 70.373,Y 79.830,Z 60.059,A 180.000,B 0.000,C 180.000} C_DIS
LIN {X 70.328,Y 79.679,Z 60.056,A 180.000,B 0.000,C 180.000} C_DIS
LIN {X 70.284,Y 79.528,Z 60.052,A 180.000,B 0.000,C 180.000} C_DIS
LIN {X 70.240,Y 79.377,Z 60.049,A 180.000,B 0.000,C 180.000} C_DIS
LIN {X 70.205,Y 79.223,Z 60.046,A 180.000,B 0.000,C 180.000} C_DIS
LIN {X 70.171,Y 79.069,Z 60.043,A 180.000,B 0.000,C 180.000} C_DIS
LIN {X 70.136,Y 78.916,Z 60.040,A 180.000,B 0.000,C 180.000} C_DIS
LIN {X 70.111,Y 78.760,Z 60.037,A 180.000,B 0.000,C 180.000} C_DIS
LIN {X 70.086,Y 78.604,Z 60.034,A 180.000,B 0.000,C 180.000} C_DIS
LIN {X 70.062,Y 78.449,Z 60.032,A 180.000,B 0.000,C 180.000} C_DIS
LIN {X 70.046,Y 78.292,Z 60.029,A 180.000,B 0.000,C 180.000} C_DIS
LIN {X 70.032,Y 78.135,Z 60.027,A 180.000,B 0.000,C 180.000} C_DIS
LIN {X 70.011,Y 77.821,Z 60.022,A 180.000,B 0.000,C 180.000} C_DIS
LIN {X 70.001,Y 77.506,Z 60.018,A 180.000,B 0.000,C 180.000} C_DIS
LIN {X 70.011,Y 77.191,Z 60.014,A 180.000,B 0.000,C 180.000} C_DIS
LIN {X 70.030,Y 76.877,Z 60.011,A 180.000,B 0.000,C 180.000} C_DIS
LIN {X 70.060,Y 76.563,Z 60.008,A 180.000,B 0.000,C 180.000} C_DIS
LIN {X 70.109,Y 76.252,Z 60.005,A 180.000,B 0.000,C 180.000} C_DIS
LIN {X 70.168,Y 75.943,Z 60.003,A 180.000,B 0.000,C 180.000} C_DIS
LIN {X 70.237,Y 75.635,Z 60.002,A 180.000,B 0.000,C 180.000} C_DIS
LIN {X 70.325,Y 75.333,Z 60.001,A 180.000,B 0.000,C 180.000} C_DIS
LIN {X 70.422,Y 75.033,Z 60.000,A 180.000,B 0.000,C 180.000} C_DIS
LIN {X 70.501,Y 74.814,Z 60.000,A 180.000,B 0.000,C 180.000} C_DIS
; Cutting Move Starts
LIN {X 70.532,Y 74.729,Z 60.000,A 180.000,B 0.000,C 180.000} C_DIS
LIN {X 70.687,Y 74.372,Z 60.000,A 180.000,B 0.000,C 180.000} C_DIS
LIN {X 70.773,Y 74.193,Z 60.000,A 180.000,B 0.000,C 180.000} C_DIS
LIN {X 70.864,Y 74.014,Z 60.000,A 180.000,B 0.000,C 180.000} C_DIS
LIN {X 70.960,Y 73.835,Z 60.000,A 180.000,B 0.000,C 180.000} C_DIS
LIN {X 71.154,Y 73.507,Z 60.000,A 180.000,B 0.000,C 180.000} C_DIS
LIN {X 71.171,Y 73.478,Z 60.000,A 180.000,B 0.000,C 180.000} C_DIS
LIN {X 71.414,Y 73.120,Z 60.000,A 180.000,B 0.000,C 180.000} C_DIS
LIN {X 71.511,Y 72.992,Z 60.000,A 180.000,B 0.000,C 180.000} C_DIS
LIN {X 71.690,Y 72.762,Z 60.000,A 180.000,B 0.000,C 180.000} C_DIS
LIN {X 71.842,Y 72.584,Z 60.000,A 180.000,B 0.000,C 180.000} C_DIS
LIN {X 72.000,Y 72.405,Z 60.000,A 180.000,B 0.000,C 180.000} C_DIS
LIN {X 72.048,Y 72.353,Z 60.000,A 180.000,B 0.000,C 180.000} C_DIS
LIN {X 72.353,Y 72.048,Z 60.000,A 180.000,B 0.000,C 180.000} C_DIS
LIN {X 72.405,Y 72.000,Z 60.000,A 180.000,B 0.000,C 180.000} C_DIS
LIN {X 72.584,Y 71.842,Z 60.000,A 180.000,B 0.000,C 180.000} C_DIS
LIN {X 72.762,Y 71.690,Z 60.000,A 180.000,B 0.000,C 180.000} C_DIS
LIN {X 72.992,Y 71.511,Z 60.000,A 180.000,B 0.000,C 180.000} C_DIS
LIN {X 73.120,Y 71.414,Z 60.000,A 180.000,B 0.000,C 180.000} C_DIS
LIN {X 73.478,Y 71.171,Z 60.000,A 180.000,B 0.000,C 180.000} C_DIS
LIN {X 73.507,Y 71.154,Z 60.000,A 180.000,B 0.000,C 180.000} C_DIS
LIN {X 73.835,Y 70.960,Z 60.000,A 180.000,B 0.000,C 180.000} C_DIS
LIN {X 74.014,Y 70.864,Z 60.000,A 180.000,B 0.000,C 180.000} C_DIS
LIN {X 74.193,Y 70.773,Z 60.000,A 180.000,B 0.000,C 180.000} C_DIS
LIN {X 74.372,Y 70.687,Z 60.000,A 180.000,B 0.000,C 180.000} C_DIS
LIN {X 74.729,Y 70.532,Z 60.000,A 180.000,B 0.000,C 180.000} C_DIS
LIN {X 74.908,Y 70.467,Z 60.000,A 180.000,B 0.000,C 180.000} C_DIS
LIN {X 75.087,Y 70.403,Z 60.000,A 180.000,B 0.000,C 180.000} C_DIS
LIN {X 75.265,Y 70.344,Z 60.000,A 180.000,B 0.000,C 180.000} C_DIS
LIN {X 75.623,Y 70.240,Z 60.000,A 180.000,B 0.000,C 180.000} C_DIS
LIN {X 75.802,Y 70.200,Z 60.000,A 180.000,B 0.000,C 180.000} C_DIS
LIN {X 75.980,Y 70.160,Z 60.000,A 180.000,B 0.000,C 180.000} C_DIS
LIN {X 76.159,Y 70.124,Z 60.000,A 180.000,B 0.000,C 180.000} C_DIS
LIN {X 76.517,Y 70.067,Z 60.000,A 180.000,B 0.000,C 180.000} C_DIS
LIN {X 76.696,Y 70.048,Z 60.000,A 180.000,B 0.000,C 180.000} C_DIS
LIN {X 76.874,Y 70.031,Z 60.000,A 180.000,B 0.000,C 180.000} C_DIS
LIN {X 77.053,Y 70.015,Z 60.000,A 180.000,B 0.000,C 180.000} C_DIS
LIN {X 77.411,Y 70.004,Z 60.000,A 180.000,B 0.000,C 180.000} C_DIS
LIN {X 77.589,Y 70.004,Z 60.000,A 180.000,B 0.000,C 180.000} C_DIS
LIN {X 77.947,Y 70.015,Z 60.000,A 180.000,B 0.000,C 180.000} C_DIS
LIN {X 78.126,Y 70.031,Z 60.000,A 180.000,B 0.000,C 180.000} C_DIS
LIN {X 78.304,Y 70.048,Z 60.000,A 180.000,B 0.000,C 180.000} C_DIS
LIN {X 78.483,Y 70.067,Z 60.000,A 180.000,B 0.000,C 180.000} C_DIS
LIN {X 78.841,Y 70.124,Z 60.000,A 180.000,B 0.000,C 180.000} C_DIS
LIN {X 79.020,Y 70.160,Z 60.000,A 180.000,B 0.000,C 180.000} C_DIS
LIN {X 79.198,Y 70.200,Z 60.000,A 180.000,B 0.000,C 180.000} C_DIS
LIN {X 79.377,Y 70.240,Z 60.000,A 180.000,B 0.000,C 180.000} C_DIS
LIN {X 79.735,Y 70.344,Z 60.000,A 180.000,B 0.000,C 180.000} C_DIS
LIN {X 79.913,Y 70.403,Z 60.000,A 180.000,B 0.000,C 180.000} C_DIS
LIN {X 80.092,Y 70.467,Z 60.000,A 180.000,B 0.000,C 180.000} C_DIS
LIN {X 80.271,Y 70.532,Z 60.000,A 180.000,B 0.000,C 180.000} C_DIS
LIN {X 80.628,Y 70.687,Z 60.000,A 180.000,B 0.000,C 180.000} C_DIS
LIN {X 80.807,Y 70.773,Z 60.000,A 180.000,B 0.000,C 180.000} C_DIS
LIN {X 80.986,Y 70.864,Z 60.000,A 180.000,B 0.000,C 180.000} C_DIS
LIN {X 81.165,Y 70.960,Z 60.000,A 180.000,B 0.000,C 180.000} C_DIS
LIN {X 81.493,Y 71.154,Z 60.000,A 180.000,B 0.000,C 180.000} C_DIS
LIN {X 81.522,Y 71.171,Z 60.000,A 180.000,B 0.000,C 180.000} C_DIS
LIN {X 81.880,Y 71.414,Z 60.000,A 180.000,B 0.000,C 180.000} C_DIS
LIN {X 82.008,Y 71.511,Z 60.000,A 180.000,B 0.000,C 180.000} C_DIS
LIN {X 82.238,Y 71.690,Z 60.000,A 180.000,B 0.000,C 180.000} C_DIS
LIN {X 82.416,Y 71.842,Z 60.000,A 180.000,B 0.000,C 180.000} C_DIS
LIN {X 82.595,Y 72.000,Z 60.000,A 180.000,B 0.000,C 180.000} C_DIS
LIN {X 82.647,Y 72.048,Z 60.000,A 180.000,B 0.000,C 180.000} C_DIS
LIN {X 82.952,Y 72.353,Z 60.000,A 180.000,B 0.000,C 180.000} C_DIS
LIN {X 83.000,Y 72.405,Z 60.000,A 180.000,B 0.000,C 180.000} C_DIS
LIN {X 83.158,Y 72.584,Z 60.000,A 180.000,B 0.000,C 180.000} C_DIS
LIN {X 83.310,Y 72.762,Z 60.000,A 180.000,B 0.000,C 180.000} C_DIS
LIN {X 83.489,Y 72.992,Z 60.000,A 180.000,B 0.000,C 180.000} C_DIS
LIN {X 83.586,Y 73.120,Z 60.000,A 180.000,B 0.000,C 180.000} C_DIS
LIN {X 83.829,Y 73.478,Z 60.000,A 180.000,B 0.000,C 180.000} C_DIS
LIN {X 83.846,Y 73.507,Z 60.000,A 180.000,B 0.000,C 180.000} C_DIS
LIN {X 84.040,Y 73.835,Z 60.000,A 180.000,B 0.000,C 180.000} C_DIS
LIN {X 84.136,Y 74.014,Z 60.000,A 180.000,B 0.000,C 180.000} C_DIS
LIN {X 84.227,Y 74.193,Z 60.000,A 180.000,B 0.000,C 180.000} C_DIS
LIN {X 84.313,Y 74.372,Z 60.000,A 180.000,B 0.000,C 180.000} C_DIS
LIN {X 84.468,Y 74.729,Z 60.000,A 180.000,B 0.000,C 180.000} C_DIS
LIN {X 84.533,Y 74.908,Z 60.000,A 180.000,B 0.000,C 180.000} C_DIS
LIN {X 84.597,Y 75.087,Z 60.000,A 180.000,B 0.000,C 180.000} C_DIS
LIN {X 84.656,Y 75.265,Z 60.000,A 180.000,B 0.000,C 180.000} C_DIS
LIN {X 84.760,Y 75.623,Z 60.000,A 180.000,B 0.000,C 180.000} C_DIS
LIN {X 84.800,Y 75.802,Z 60.000,A 180.000,B 0.000,C 180.000} C_DIS
LIN {X 84.840,Y 75.980,Z 60.000,A 180.000,B 0.000,C 180.000} C_DIS
LIN {X 84.876,Y 76.159,Z 60.000,A 180.000,B 0.000,C 180.000} C_DIS
LIN {X 84.933,Y 76.517,Z 60.000,A 180.000,B 0.000,C 180.000} C_DIS
LIN {X 84.952,Y 76.696,Z 60.000,A 180.000,B 0.000,C 180.000} C_DIS
LIN {X 84.969,Y 76.874,Z 60.000,A 180.000,B 0.000,C 180.000} C_DIS
LIN {X 84.985,Y 77.053,Z 60.000,A 180.000,B 0.000,C 180.000} C_DIS
LIN {X 84.996,Y 77.411,Z 60.000,A 180.000,B 0.000,C 180.000} C_DIS
LIN {X 84.996,Y 77.589,Z 60.000,A 180.000,B 0.000,C 180.000} C_DIS
LIN {X 84.985,Y 77.947,Z 60.000,A 180.000,B 0.000,C 180.000} C_DIS
LIN {X 84.969,Y 78.126,Z 60.000,A 180.000,B 0.000,C 180.000} C_DIS
LIN {X 84.952,Y 78.304,Z 60.000,A 180.000,B 0.000,C 180.000} C_DIS
LIN {X 84.933,Y 78.483,Z 60.000,A 180.000,B 0.000,C 180.000} C_DIS
LIN {X 84.876,Y 78.841,Z 60.000,A 180.000,B 0.000,C 180.000} C_DIS
LIN {X 84.840,Y 79.020,Z 60.000,A 180.000,B 0.000,C 180.000} C_DIS
LIN {X 84.800,Y 79.198,Z 60.000,A 180.000,B 0.000,C 180.000} C_DIS
LIN {X 84.760,Y 79.377,Z 60.000,A 180.000,B 0.000,C 180.000} C_DIS
LIN {X 84.656,Y 79.735,Z 60.000,A 180.000,B 0.000,C 180.000} C_DIS
LIN {X 84.597,Y 79.913,Z 60.000,A 180.000,B 0.000,C 180.000} C_DIS
LIN {X 84.533,Y 80.092,Z 60.000,A 180.000,B 0.000,C 180.000} C_DIS
LIN {X 84.468,Y 80.271,Z 60.000,A 180.000,B 0.000,C 180.000} C_DIS
LIN {X 84.313,Y 80.628,Z 60.000,A 180.000,B 0.000,C 180.000} C_DIS
LIN {X 84.227,Y 80.807,Z 60.000,A 180.000,B 0.000,C 180.000} C_DIS
LIN {X 84.136,Y 80.986,Z 60.000,A 180.000,B 0.000,C 180.000} C_DIS
LIN {X 84.040,Y 81.165,Z 60.000,A 180.000,B 0.000,C 180.000} C_DIS
LIN {X 83.846,Y 81.493,Z 60.000,A 180.000,B 0.000,C 180.000} C_DIS
LIN {X 83.829,Y 81.522,Z 60.000,A 180.000,B 0.000,C 180.000} C_DIS
LIN {X 83.586,Y 81.880,Z 60.000,A 180.000,B 0.000,C 180.000} C_DIS
LIN {X 83.489,Y 82.008,Z 60.000,A 180.000,B 0.000,C 180.000} C_DIS
LIN {X 83.310,Y 82.238,Z 60.000,A 180.000,B 0.000,C 180.000} C_DIS
LIN {X 83.158,Y 82.416,Z 60.000,A 180.000,B 0.000,C 180.000} C_DIS
LIN {X 83.000,Y 82.595,Z 60.000,A 180.000,B 0.000,C 180.000} C_DIS
LIN {X 82.952,Y 82.647,Z 60.000,A 180.000,B 0.000,C 180.000} C_DIS
LIN {X 82.647,Y 82.952,Z 60.000,A 180.000,B 0.000,C 180.000} C_DIS
LIN {X 82.595,Y 83.000,Z 60.000,A 180.000,B 0.000,C 180.000} C_DIS
LIN {X 82.416,Y 83.158,Z 60.000,A 180.000,B 0.000,C 180.000} C_DIS
LIN {X 82.238,Y 83.310,Z 60.000,A 180.000,B 0.000,C 180.000} C_DIS
LIN {X 82.008,Y 83.489,Z 60.000,A 180.000,B 0.000,C 180.000} C_DIS
LIN {X 81.880,Y 83.586,Z 60.000,A 180.000,B 0.000,C 180.000} C_DIS
LIN {X 81.522,Y 83.829,Z 60.000,A 180.000,B 0.000,C 180.000} C_DIS
LIN {X 81.493,Y 83.846,Z 60.000,A 180.000,B 0.000,C 180.000} C_DIS
LIN {X 81.165,Y 84.040,Z 60.000,A 180.000,B 0.000,C 180.000} C_DIS
LIN {X 80.986,Y 84.136,Z 60.000,A 180.000,B 0.000,C 180.000} C_DIS
LIN {X 80.807,Y 84.227,Z 60.000,A 180.000,B 0.000,C 180.000} C_DIS
LIN {X 80.628,Y 84.313,Z 60.000,A 180.000,B 0.000,C 180.000} C_DIS
LIN {X 80.271,Y 84.468,Z 60.000,A 180.000,B 0.000,C 180.000} C_DIS
LIN {X 80.092,Y 84.533,Z 60.000,A 180.000,B 0.000,C 180.000} C_DIS
LIN {X 79.913,Y 84.597,Z 60.000,A 180.000,B 0.000,C 180.000} C_DIS
LIN {X 79.735,Y 84.656,Z 60.000,A 180.000,B 0.000,C 180.000} C_DIS
LIN {X 79.377,Y 84.760,Z 60.000,A 180.000,B 0.000,C 180.000} C_DIS
LIN {X 79.198,Y 84.800,Z 60.000,A 180.000,B 0.000,C 180.000} C_DIS
LIN {X 79.020,Y 84.840,Z 60.000,A 180.000,B 0.000,C 180.000} C_DIS
LIN {X 78.841,Y 84.876,Z 60.000,A 180.000,B 0.000,C 180.000} C_DIS
LIN {X 78.483,Y 84.933,Z 60.000,A 180.000,B 0.000,C 180.000} C_DIS
LIN {X 78.304,Y 84.952,Z 60.000,A 180.000,B 0.000,C 180.000} C_DIS
LIN {X 78.126,Y 84.969,Z 60.000,A 180.000,B 0.000,C 180.000} C_DIS
LIN {X 77.947,Y 84.985,Z 60.000,A 180.000,B 0.000,C 180.000} C_DIS
LIN {X 77.589,Y 84.996,Z 60.000,A 180.000,B 0.000,C 180.000} C_DIS
LIN {X 77.411,Y 84.996,Z 60.000,A 180.000,B 0.000,C 180.000} C_DIS
LIN {X 77.053,Y 84.985,Z 60.000,A 180.000,B 0.000,C 180.000} C_DIS
LIN {X 76.874,Y 84.969,Z 60.000,A 180.000,B 0.000,C 180.000} C_DIS
LIN {X 76.696,Y 84.952,Z 60.000,A 180.000,B 0.000,C 180.000} C_DIS
LIN {X 76.517,Y 84.933,Z 60.000,A 180.000,B 0.000,C 180.000} C_DIS
LIN {X 76.159,Y 84.876,Z 60.000,A 180.000,B 0.000,C 180.000} C_DIS
LIN {X 75.980,Y 84.840,Z 60.000,A 180.000,B 0.000,C 180.000} C_DIS
LIN {X 75.802,Y 84.800,Z 60.000,A 180.000,B 0.000,C 180.000} C_DIS
LIN {X 75.623,Y 84.760,Z 60.000,A 180.000,B 0.000,C 180.000} C_DIS
LIN {X 75.265,Y 84.656,Z 60.000,A 180.000,B 0.000,C 180.000} C_DIS
LIN {X 75.087,Y 84.597,Z 60.000,A 180.000,B 0.000,C 180.000} C_DIS
LIN {X 74.908,Y 84.533,Z 60.000,A 180.000,B 0.000,C 180.000} C_DIS
LIN {X 74.729,Y 84.468,Z 60.000,A 180.000,B 0.000,C 180.000} C_DIS
LIN {X 74.372,Y 84.313,Z 60.000,A 180.000,B 0.000,C 180.000} C_DIS
LIN {X 74.193,Y 84.227,Z 60.000,A 180.000,B 0.000,C 180.000} C_DIS
LIN {X 74.014,Y 84.136,Z 60.000,A 180.000,B 0.000,C 180.000} C_DIS
LIN {X 73.835,Y 84.040,Z 60.000,A 180.000,B 0.000,C 180.000} C_DIS
LIN {X 73.507,Y 83.846,Z 60.000,A 180.000,B 0.000,C 180.000} C_DIS
LIN {X 73.478,Y 83.829,Z 60.000,A 180.000,B 0.000,C 180.000} C_DIS
LIN {X 73.120,Y 83.586,Z 60.000,A 180.000,B 0.000,C 180.000} C_DIS
LIN {X 72.992,Y 83.489,Z 60.000,A 180.000,B 0.000,C 180.000} C_DIS
LIN {X 72.762,Y 83.310,Z 60.000,A 180.000,B 0.000,C 180.000} C_DIS
LIN {X 72.584,Y 83.158,Z 60.000,A 180.000,B 0.000,C 180.000} C_DIS
LIN {X 72.405,Y 83.000,Z 60.000,A 180.000,B 0.000,C 180.000} C_DIS
LIN {X 72.353,Y 82.952,Z 60.000,A 180.000,B 0.000,C 180.000} C_DIS
LIN {X 72.048,Y 82.647,Z 60.000,A 180.000,B 0.000,C 180.000} C_DIS
LIN {X 72.000,Y 82.595,Z 60.000,A 180.000,B 0.000,C 180.000} C_DIS
LIN {X 71.842,Y 82.416,Z 60.000,A 180.000,B 0.000,C 180.000} C_DIS
LIN {X 71.690,Y 82.238,Z 60.000,A 180.000,B 0.000,C 180.000} C_DIS
LIN {X 71.511,Y 82.008,Z 60.000,A 180.000,B 0.000,C 180.000} C_DIS
LIN {X 71.414,Y 81.880,Z 60.000,A 180.000,B 0.000,C 180.000} C_DIS
LIN {X 71.171,Y 81.522,Z 60.000,A 180.000,B 0.000,C 180.000} C_DIS
LIN {X 71.154,Y 81.493,Z 60.000,A 180.000,B 0.000,C 180.000} C_DIS
LIN {X 70.960,Y 81.165,Z 60.000,A 180.000,B 0.000,C 180.000} C_DIS
LIN {X 70.864,Y 80.986,Z 60.000,A 180.000,B 0.000,C 180.000} C_DIS
LIN {X 70.773,Y 80.807,Z 60.000,A 180.000,B 0.000,C 180.000} C_DIS
LIN {X 70.687,Y 80.628,Z 60.000,A 180.000,B 0.000,C 180.000} C_DIS
LIN {X 70.532,Y 80.271,Z 60.000,A 180.000,B 0.000,C 180.000} C_DIS
LIN {X 70.467,Y 80.092,Z 60.000,A 180.000,B 0.000,C 180.000} C_DIS
LIN {X 70.403,Y 79.913,Z 60.000,A 180.000,B 0.000,C 180.000} C_DIS
LIN {X 70.344,Y 79.735,Z 60.000,A 180.000,B 0.000,C 180.000} C_DIS
LIN {X 70.240,Y 79.377,Z 60.000,A 180.000,B 0.000,C 180.000} C_DIS
LIN {X 70.200,Y 79.198,Z 60.000,A 180.000,B 0.000,C 180.000} C_DIS
LIN {X 70.160,Y 79.020,Z 60.000,A 180.000,B 0.000,C 180.000} C_DIS
LIN {X 70.124,Y 78.841,Z 60.000,A 180.000,B 0.000,C 180.000} C_DIS
LIN {X 70.067,Y 78.483,Z 60.000,A 180.000,B 0.000,C 180.000} C_DIS
LIN {X 70.048,Y 78.304,Z 60.000,A 180.000,B 0.000,C 180.000} C_DIS
LIN {X 70.031,Y 78.126,Z 60.000,A 180.000,B 0.000,C 180.000} C_DIS
LIN {X 70.015,Y 77.947,Z 60.000,A 180.000,B 0.000,C 180.000} C_DIS
LIN {X 70.004,Y 77.589,Z 60.000,A 180.000,B 0.000,C 180.000} C_DIS
LIN {X 70.004,Y 77.411,Z 60.000,A 180.000,B 0.000,C 180.000} C_DIS
LIN {X 70.015,Y 77.053,Z 60.000,A 180.000,B 0.000,C 180.000} C_DIS
LIN {X 70.031,Y 76.874,Z 60.000,A 180.000,B 0.000,C 180.000} C_DIS
LIN {X 70.048,Y 76.696,Z 60.000,A 180.000,B 0.000,C 180.000} C_DIS
LIN {X 70.067,Y 76.517,Z 60.000,A 180.000,B 0.000,C 180.000} C_DIS
LIN {X 70.124,Y 76.159,Z 60.000,A 180.000,B 0.000,C 180.000} C_DIS
LIN {X 70.160,Y 75.980,Z 60.000,A 180.000,B 0.000,C 180.000} C_DIS
LIN {X 70.200,Y 75.802,Z 60.000,A 180.000,B 0.000,C 180.000} C_DIS
LIN {X 70.240,Y 75.623,Z 60.000,A 180.000,B 0.000,C 180.000} C_DIS
LIN {X 70.344,Y 75.265,Z 60.000,A 180.000,B 0.000,C 180.000} C_DIS
LIN {X 70.403,Y 75.087,Z 60.000,A 180.000,B 0.000,C 180.000} C_DIS
LIN {X 70.467,Y 74.908,Z 60.000,A 180.000,B 0.000,C 180.000} C_DIS
LIN {X 70.501,Y 74.814,Z 60.000,A 180.000,B 0.000,C 180.000} C_DIS
; Link Move Starts
LIN {X 70.621,Y 74.523,Z 60.000,A 180.000,B 0.000,C 180.000} C_DIS
LIN {X 70.751,Y 74.236,Z 59.999,A 180.000,B 0.000,C 180.000} C_DIS
LIN {X 70.894,Y 73.956,Z 59.998,A 180.000,B 0.000,C 180.000} C_DIS
LIN {X 71.050,Y 73.682,Z 59.996,A 180.000,B 0.000,C 180.000} C_DIS
LIN {X 71.215,Y 73.414,Z 59.994,A 180.000,B 0.000,C 180.000} C_DIS
LIN {X 71.392,Y 73.153,Z 59.991,A 180.000,B 0.000,C 180.000} C_DIS
LIN {X 71.581,Y 72.901,Z 59.988,A 180.000,B 0.000,C 180.000} C_DIS
LIN {X 71.779,Y 72.656,Z 59.985,A 180.000,B 0.000,C 180.000} C_DIS
LIN {X 71.987,Y 72.420,Z 59.981,A 180.000,B 0.000,C 180.000} C_DIS
LIN {X 72.206,Y 72.194,Z 59.977,A 180.000,B 0.000,C 180.000} C_DIS
LIN {X 72.433,Y 71.975,Z 59.972,A 180.000,B 0.000,C 180.000} C_DIS
LIN {X 72.551,Y 71.871,Z 59.969,A 180.000,B 0.000,C 180.000} C_DIS
LIN {X 72.669,Y 71.767,Z 59.967,A 180.000,B 0.000,C 180.000} C_DIS
LIN {X 72.791,Y 71.667,Z 59.964,A 180.000,B 0.000,C 180.000} C_DIS
LIN {X 72.916,Y 71.570,Z 59.961,A 180.000,B 0.000,C 180.000} C_DIS
LIN {X 73.040,Y 71.474,Z 59.959,A 180.000,B 0.000,C 180.000} C_DIS
LIN {X 73.168,Y 71.382,Z 59.956,A 180.000,B 0.000,C 180.000} C_DIS
LIN {X 73.298,Y 71.293,Z 59.952,A 180.000,B 0.000,C 180.000} C_DIS
LIN {X 73.428,Y 71.205,Z 59.949,A 180.000,B 0.000,C 180.000} C_DIS
LIN {X 73.562,Y 71.121,Z 59.946,A 180.000,B 0.000,C 180.000} C_DIS
LIN {X 73.697,Y 71.041,Z 59.943,A 180.000,B 0.000,C 180.000} C_DIS
LIN {X 73.833,Y 70.961,Z 59.939,A 180.000,B 0.000,C 180.000} C_DIS
LIN {X 73.971,Y 70.886,Z 59.936,A 180.000,B 0.000,C 180.000} C_DIS
LIN {X 74.112,Y 70.814,Z 59.932,A 180.000,B 0.000,C 180.000} C_DIS
LIN {X 74.252,Y 70.743,Z 59.928,A 180.000,B 0.000,C 180.000} C_DIS
LIN {X 74.395,Y 70.677,Z 59.925,A 180.000,B 0.000,C 180.000} C_DIS
LIN {X 74.540,Y 70.614,Z 59.921,A 180.000,B 0.000,C 180.000} C_DIS
LIN {X 74.684,Y 70.552,Z 59.917,A 180.000,B 0.000,C 180.000} C_DIS
LIN {X 74.831,Y 70.495,Z 59.913,A 180.000,B 0.000,C 180.000} C_DIS
LIN {X 74.979,Y 70.442,Z 59.909,A 180.000,B 0.000,C 180.000} C_DIS
LIN {X 75.127,Y 70.388,Z 59.905,A 180.000,B 0.000,C 180.000} C_DIS
LIN {X 75.278,Y 70.341,Z 59.900,A 180.000,B 0.000,C 180.000} C_DIS
LIN {X 75.429,Y 70.297,Z 59.896,A 180.000,B 0.000,C 180.000} C_DIS
LIN {X 75.580,Y 70.253,Z 59.892,A 180.000,B 0.000,C 180.000} C_DIS
LIN {X 75.733,Y 70.215,Z 59.887,A 180.000,B 0.000,C 180.000} C_DIS
LIN {X 75.887,Y 70.181,Z 59.883,A 180.000,B 0.000,C 180.000} C_DIS
LIN {X 76.040,Y 70.146,Z 59.878,A 180.000,B 0.000,C 180.000} C_DIS
LIN {X 76.195,Y 70.118,Z 59.873,A 180.000,B 0.000,C 180.000} C_DIS
LIN {X 76.351,Y 70.094,Z 59.869,A 180.000,B 0.000,C 180.000} C_DIS
LIN {X 76.506,Y 70.069,Z 59.864,A 180.000,B 0.000,C 180.000} C_DIS
LIN {X 76.663,Y 70.051,Z 59.859,A 180.000,B 0.000,C 180.000} C_DIS
LIN {X 76.820,Y 70.036,Z 59.854,A 180.000,B 0.000,C 180.000} C_DIS
LIN {X 76.898,Y 70.028,Z 59.851,A 180.000,B 0.000,C 180.000} C_DIS
LIN {X 76.976,Y 70.021,Z 59.849,A 180.000,B 0.000,C 180.000} C_DIS
LIN {X 77.055,Y 70.015,Z 59.846,A 180.000,B 0.000,C 180.000} C_DIS
LIN {X 77.134,Y 70.013,Z 59.844,A 180.000,B 0.000,C 180.000} C_DIS
LIN {X 77.212,Y 70.010,Z 59.841,A 180.000,B 0.000,C 180.000} C_DIS
LIN {X 77.370,Y 70.005,Z 59.836,A 180.000,B 0.000,C 180.000} C_DIS
LIN {X 77.449,Y 70.003,Z 59.833,A 180.000,B 0.000,C 180.000} C_DIS
LIN {X 77.527,Y 70.002,Z 59.831,A 180.000,B 0.000,C 180.000} C_DIS
LIN {X 77.606,Y 70.005,Z 59.828,A 180.000,B 0.000,C 180.000} C_DIS
LIN {X 77.763,Y 70.010,Z 59.823,A 180.000,B 0.000,C 180.000} C_DIS
LIN {X 77.921,Y 70.014,Z 59.817,A 180.000,B 0.000,C 180.000} C_DIS
LIN {X 78.000,Y 70.019,Z 59.815,A 180.000,B 0.000,C 180.000} C_DIS
LIN {X 78.156,Y 70.034,Z 59.809,A 180.000,B 0.000,C 180.000} C_DIS
LIN {X 78.235,Y 70.041,Z 59.806,A 180.000,B 0.000,C 180.000} C_DIS
LIN {X 78.392,Y 70.056,Z 59.801,A 180.000,B 0.000,C 180.000} C_DIS
LIN {X 78.470,Y 70.065,Z 59.798,A 180.000,B 0.000,C 180.000} C_DIS
LIN {X 78.548,Y 70.077,Z 59.796,A 180.000,B 0.000,C 180.000} C_DIS
LIN {X 78.703,Y 70.102,Z 59.790,A 180.000,B 0.000,C 180.000} C_DIS
LIN {X 78.859,Y 70.127,Z 59.785,A 180.000,B 0.000,C 180.000} C_DIS
LIN {X 78.936,Y 70.141,Z 59.782,A 180.000,B 0.000,C 180.000} C_DIS
LIN {X 79.090,Y 70.175,Z 59.776,A 180.000,B 0.000,C 180.000} C_DIS
LIN {X 79.167,Y 70.193,Z 59.774,A 180.000,B 0.000,C 180.000} C_DIS
LIN {X 79.320,Y 70.227,Z 59.768,A 180.000,B 0.000,C 180.000} C_DIS
LIN {X 79.397,Y 70.246,Z 59.765,A 180.000,B 0.000,C 180.000} C_DIS
LIN {X 79.472,Y 70.268,Z 59.763,A 180.000,B 0.000,C 180.000} C_DIS
LIN {X 79.624,Y 70.312,Z 59.757,A 180.000,B 0.000,C 180.000} C_DIS
LIN {X 79.775,Y 70.356,Z 59.752,A 180.000,B 0.000,C 180.000} C_DIS
LIN {X 79.850,Y 70.380,Z 59.749,A 180.000,B 0.000,C 180.000} C_DIS
LIN {X 79.998,Y 70.433,Z 59.743,A 180.000,B 0.000,C 180.000} C_DIS
LIN {X 80.072,Y 70.460,Z 59.741,A 180.000,B 0.000,C 180.000} C_DIS
LIN {X 80.220,Y 70.513,Z 59.735,A 180.000,B 0.000,C 180.000} C_DIS
LIN {X 80.294,Y 70.542,Z 59.732,A 180.000,B 0.000,C 180.000} C_DIS
LIN {X 80.366,Y 70.573,Z 59.730,A 180.000,B 0.000,C 180.000} C_DIS
LIN {X 80.510,Y 70.636,Z 59.724,A 180.000,B 0.000,C 180.000} C_DIS
LIN {X 80.655,Y 70.699,Z 59.719,A 180.000,B 0.000,C 180.000} C_DIS
LIN {X 80.726,Y 70.732,Z 59.716,A 180.000,B 0.000,C 180.000} C_DIS
LIN {X 80.867,Y 70.804,Z 59.710,A 180.000,B 0.000,C 180.000} C_DIS
LIN {X 80.937,Y 70.839,Z 59.708,A 180.000,B 0.000,C 180.000} C_DIS
LIN {X 81.077,Y 70.911,Z 59.702,A 180.000,B 0.000,C 180.000} C_DIS
LIN {X 81.146,Y 70.949,Z 59.699,A 180.000,B 0.000,C 180.000} C_DIS
LIN {X 81.214,Y 70.989,Z 59.697,A 180.000,B 0.000,C 180.000} C_DIS
LIN {X 81.350,Y 71.069,Z 59.691,A 180.000,B 0.000,C 180.000} C_DIS
LIN {X 81.485,Y 71.149,Z 59.686,A 180.000,B 0.000,C 180.000} C_DIS
LIN {X 81.552,Y 71.191,Z 59.683,A 180.000,B 0.000,C 180.000} C_DIS
LIN {X 81.682,Y 71.280,Z 59.677,A 180.000,B 0.000,C 180.000} C_DIS
LIN {X 81.747,Y 71.324,Z 59.675,A 180.000,B 0.000,C 180.000} C_DIS
LIN {X 81.877,Y 71.413,Z 59.669,A 180.000,B 0.000,C 180.000} C_DIS
LIN {X 81.941,Y 71.459,Z 59.666,A 180.000,B 0.000,C 180.000} C_DIS
LIN {X 82.065,Y 71.556,Z 59.661,A 180.000,B 0.000,C 180.000} C_DIS
LIN {X 82.252,Y 71.700,Z 59.653,A 180.000,B 0.000,C 180.000} C_DIS
LIN {X 82.313,Y 71.751,Z 59.650,A 180.000,B 0.000,C 180.000} C_DIS
LIN {X 82.608,Y 72.011,Z 59.636,A 180.000,B 0.000,C 180.000} C_DIS
LIN {X 82.665,Y 72.065,Z 59.633,A 180.000,B 0.000,C 180.000} C_DIS
LIN {X 82.776,Y 72.177,Z 59.628,A 180.000,B 0.000,C 180.000} C_DIS
LIN {X 82.943,Y 72.344,Z 59.620,A 180.000,B 0.000,C 180.000} C_DIS
LIN {X 82.997,Y 72.402,Z 59.617,A 180.000,B 0.000,C 180.000} C_DIS
LIN {X 83.257,Y 72.697,Z 59.603,A 180.000,B 0.000,C 180.000} C_DIS
LIN {X 83.307,Y 72.758,Z 59.600,A 180.000,B 0.000,C 180.000} C_DIS
LIN {X 83.549,Y 73.069,Z 59.587,A 180.000,B 0.000,C 180.000} C_DIS
LIN {X 83.594,Y 73.133,Z 59.584,A 180.000,B 0.000,C 180.000} C_DIS
LIN {X 83.816,Y 73.459,Z 59.570,A 180.000,B 0.000,C 180.000} C_DIS
LIN {X 83.857,Y 73.526,Z 59.567,A 180.000,B 0.000,C 180.000} C_DIS
LIN {X 84.058,Y 73.865,Z 59.554,A 180.000,B 0.000,C 180.000} C_DIS
LIN {X 84.095,Y 73.934,Z 59.551,A 180.000,B 0.000,C 180.000} C_DIS
LIN {X 84.274,Y 74.285,Z 59.537,A 180.000,B 0.000,C 180.000} C_DIS
LIN {X 84.306,Y 74.357,Z 59.534,A 180.000,B 0.000,C 180.000} C_DIS
LIN {X 84.463,Y 74.718,Z 59.521,A 180.000,B 0.000,C 180.000} C_DIS
LIN {X 84.491,Y 74.792,Z 59.518,A 180.000,B 0.000,C 180.000} C_DIS
LIN {X 84.624,Y 75.162,Z 59.504,A 180.000,B 0.000,C 180.000} C_DIS
LIN {X 84.648,Y 75.237,Z 59.501,A 180.000,B 0.000,C 180.000} C_DIS
LIN {X 84.757,Y 75.615,Z 59.488,A 180.000,B 0.000,C 180.000} C_DIS
LIN {X 84.776,Y 75.692,Z 59.485,A 180.000,B 0.000,C 180.000} C_DIS
LIN {X 84.862,Y 76.076,Z 59.471,A 180.000,B 0.000,C 180.000} C_DIS
LIN {X 84.875,Y 76.154,Z 59.468,A 180.000,B 0.000,C 180.000} C_DIS
LIN {X 84.937,Y 76.543,Z 59.455,A 180.000,B 0.000,C 180.000} C_DIS
LIN {X 84.945,Y 76.621,Z 59.452,A 180.000,B 0.000,C 180.000} C_DIS
LIN {X 84.982,Y 77.013,Z 59.438,A 180.000,B 0.000,C 180.000} C_DIS
LIN {X 84.986,Y 77.092,Z 59.435,A 180.000,B 0.000,C 180.000} C_DIS
LIN {X 84.998,Y 77.485,Z 59.422,A 180.000,B 0.000,C 180.000} C_DIS
LIN {X 84.997,Y 77.564,Z 59.419,A 180.000,B 0.000,C 180.000} C_DIS
LIN {X 84.984,Y 77.958,Z 59.405,A 180.000,B 0.000,C 180.000} C_DIS
LIN {X 84.978,Y 78.036,Z 59.402,A 180.000,B 0.000,C 180.000} C_DIS
LIN {X 84.963,Y 78.193,Z 59.397,A 180.000,B 0.000,C 180.000} C_DIS
LIN {X 84.941,Y 78.428,Z 59.389,A 180.000,B 0.000,C 180.000} C_DIS
LIN {X 84.929,Y 78.506,Z 59.386,A 180.000,B 0.000,C 180.000} C_DIS
LIN {X 84.868,Y 78.895,Z 59.372,A 180.000,B 0.000,C 180.000} C_DIS
LIN {X 84.851,Y 78.972,Z 59.369,A 180.000,B 0.000,C 180.000} C_DIS
LIN {X 84.817,Y 79.126,Z 59.364,A 180.000,B 0.000,C 180.000} C_DIS
LIN {X 84.765,Y 79.356,Z 59.356,A 180.000,B 0.000,C 180.000} C_DIS
LIN {X 84.744,Y 79.432,Z 59.353,A 180.000,B 0.000,C 180.000} C_DIS
LIN {X 84.634,Y 79.810,Z 59.339,A 180.000,B 0.000,C 180.000} C_DIS
LIN {X 84.608,Y 79.885,Z 59.336,A 180.000,B 0.000,C 180.000} C_DIS
LIN {X 84.581,Y 79.959,Z 59.334,A 180.000,B 0.000,C 180.000} C_DIS
LIN {X 84.528,Y 80.107,Z 59.328,A 180.000,B 0.000,C 180.000} C_DIS
LIN {X 84.474,Y 80.255,Z 59.323,A 180.000,B 0.000,C 180.000} C_DIS
LIN {X 84.443,Y 80.327,Z 59.320,A 180.000,B 0.000,C 180.000} C_DIS
LIN {X 84.381,Y 80.472,Z 59.314,A 180.000,B 0.000,C 180.000} C_DIS
LIN {X 84.349,Y 80.544,Z 59.312,A 180.000,B 0.000,C 180.000} C_DIS
LIN {X 84.287,Y 80.689,Z 59.306,A 180.000,B 0.000,C 180.000} C_DIS
LIN {X 84.251,Y 80.759,Z 59.303,A 180.000,B 0.000,C 180.000} C_DIS
LIN {X 84.216,Y 80.829,Z 59.301,A 180.000,B 0.000,C 180.000} C_DIS
LIN {X 84.144,Y 80.970,Z 59.295,A 180.000,B 0.000,C 180.000} C_DIS
LIN {X 84.073,Y 81.110,Z 59.290,A 180.000,B 0.000,C 180.000} C_DIS
LIN {X 84.033,Y 81.178,Z 59.287,A 180.000,B 0.000,C 180.000} C_DIS
LIN {X 83.952,Y 81.313,Z 59.281,A 180.000,B 0.000,C 180.000} C_DIS
LIN {X 83.912,Y 81.381,Z 59.279,A 180.000,B 0.000,C 180.000} C_DIS
LIN {X 83.832,Y 81.517,Z 59.273,A 180.000,B 0.000,C 180.000} C_DIS
LIN {X 83.788,Y 81.582,Z 59.270,A 180.000,B 0.000,C 180.000} C_DIS
LIN {X 83.744,Y 81.647,Z 59.268,A 180.000,B 0.000,C 180.000} C_DIS
LIN {X 83.655,Y 81.777,Z 59.262,A 180.000,B 0.000,C 180.000} C_DIS
LIN {X 83.567,Y 81.908,Z 59.257,A 180.000,B 0.000,C 180.000} C_DIS
LIN {X 83.470,Y 82.032,Z 59.251,A 180.000,B 0.000,C 180.000} C_DIS
LIN {X 83.325,Y 82.219,Z 59.243,A 180.000,B 0.000,C 180.000} C_DIS
LIN {X 83.277,Y 82.281,Z 59.240,A 180.000,B 0.000,C 180.000} C_DIS
LIN {X 83.121,Y 82.458,Z 59.232,A 180.000,B 0.000,C 180.000} C_DIS
LIN {X 83.016,Y 82.576,Z 59.226,A 180.000,B 0.000,C 180.000} C_DIS
LIN {X 82.964,Y 82.635,Z 59.224,A 180.000,B 0.000,C 180.000} C_DIS
LIN {X 82.853,Y 82.747,Z 59.218,A 180.000,B 0.000,C 180.000} C_DIS
LIN {X 82.686,Y 82.914,Z 59.210,A 180.000,B 0.000,C 180.000} C_DIS
LIN {X 82.630,Y 82.969,Z 59.207,A 180.000,B 0.000,C 180.000} C_DIS
LIN {X 82.453,Y 83.126,Z 59.199,A 180.000,B 0.000,C 180.000} C_DIS
LIN {X 82.335,Y 83.230,Z 59.193,A 180.000,B 0.000,C 180.000} C_DIS
LIN {X 82.275,Y 83.282,Z 59.191,A 180.000,B 0.000,C 180.000} C_DIS
LIN {X 82.151,Y 83.378,Z 59.185,A 180.000,B 0.000,C 180.000} C_DIS
LIN {X 82.026,Y 83.475,Z 59.180,A 180.000,B 0.000,C 180.000} C_DIS
LIN {X 81.964,Y 83.523,Z 59.177,A 180.000,B 0.000,C 180.000} C_DIS
LIN {X 81.902,Y 83.571,Z 59.174,A 180.000,B 0.000,C 180.000} C_DIS
LIN {X 81.771,Y 83.659,Z 59.169,A 180.000,B 0.000,C 180.000} C_DIS
LIN {X 81.641,Y 83.748,Z 59.164,A 180.000,B 0.000,C 180.000} C_DIS
LIN {X 81.576,Y 83.792,Z 59.161,A 180.000,B 0.000,C 180.000} C_DIS
LIN {X 81.510,Y 83.836,Z 59.159,A 180.000,B 0.000,C 180.000} C_DIS
LIN {X 81.443,Y 83.876,Z 59.156,A 180.000,B 0.000,C 180.000} C_DIS
LIN {X 81.375,Y 83.916,Z 59.154,A 180.000,B 0.000,C 180.000} C_DIS
LIN {X 81.307,Y 83.956,Z 59.151,A 180.000,B 0.000,C 180.000} C_DIS
LIN {X 81.239,Y 83.996,Z 59.149,A 180.000,B 0.000,C 180.000} C_DIS
LIN {X 81.103,Y 84.076,Z 59.144,A 180.000,B 0.000,C 180.000} C_DIS
LIN {X 80.963,Y 84.147,Z 59.139,A 180.000,B 0.000,C 180.000} C_DIS
LIN {X 80.823,Y 84.219,Z 59.134,A 180.000,B 0.000,C 180.000} C_DIS
LIN {X 80.682,Y 84.290,Z 59.129,A 180.000,B 0.000,C 180.000} C_DIS
LIN {X 80.537,Y 84.352,Z 59.124,A 180.000,B 0.000,C 180.000} C_DIS
LIN {X 80.393,Y 84.415,Z 59.120,A 180.000,B 0.000,C 180.000} C_DIS
LIN {X 80.248,Y 84.477,Z 59.115,A 180.000,B 0.000,C 180.000} C_DIS
LIN {X 80.100,Y 84.530,Z 59.111,A 180.000,B 0.000,C 180.000} C_DIS
LIN {X 79.952,Y 84.583,Z 59.106,A 180.000,B 0.000,C 180.000} C_DIS
LIN {X 79.803,Y 84.636,Z 59.102,A 180.000,B 0.000,C 180.000} C_DIS
LIN {X 79.652,Y 84.680,Z 59.097,A 180.000,B 0.000,C 180.000} C_DIS
LIN {X 79.501,Y 84.724,Z 59.093,A 180.000,B 0.000,C 180.000} C_DIS
LIN {X 79.349,Y 84.767,Z 59.089,A 180.000,B 0.000,C 180.000} C_DIS
LIN {X 79.195,Y 84.801,Z 59.085,A 180.000,B 0.000,C 180.000} C_DIS
LIN {X 79.042,Y 84.835,Z 59.081,A 180.000,B 0.000,C 180.000} C_DIS
LIN {X 78.888,Y 84.869,Z 59.077,A 180.000,B 0.000,C 180.000} C_DIS
LIN {X 78.732,Y 84.893,Z 59.073,A 180.000,B 0.000,C 180.000} C_DIS
LIN {X 78.576,Y 84.918,Z 59.070,A 180.000,B 0.000,C 180.000} C_DIS
LIN {X 78.421,Y 84.941,Z 59.066,A 180.000,B 0.000,C 180.000} C_DIS
LIN {X 78.264,Y 84.956,Z 59.062,A 180.000,B 0.000,C 180.000} C_DIS
LIN {X 78.107,Y 84.971,Z 59.059,A 180.000,B 0.000,C 180.000} C_DIS
LIN {X 77.950,Y 84.985,Z 59.056,A 180.000,B 0.000,C 180.000} C_DIS
LIN {X 77.793,Y 84.990,Z 59.052,A 180.000,B 0.000,C 180.000} C_DIS
LIN {X 77.635,Y 84.995,Z 59.049,A 180.000,B 0.000,C 180.000} C_DIS
LIN {X 77.478,Y 84.998,Z 59.046,A 180.000,B 0.000,C 180.000} C_DIS
LIN {X 77.320,Y 84.993,Z 59.043,A 180.000,B 0.000,C 180.000} C_DIS
LIN {X 77.163,Y 84.988,Z 59.040,A 180.000,B 0.000,C 180.000} C_DIS
LIN {X 77.006,Y 84.982,Z 59.037,A 180.000,B 0.000,C 180.000} C_DIS
LIN {X 76.849,Y 84.967,Z 59.034,A 180.000,B 0.000,C 180.000} C_DIS
LIN {X 76.692,Y 84.952,Z 59.032,A 180.000,B 0.000,C 180.000} C_DIS
LIN {X 76.535,Y 84.936,Z 59.029,A 180.000,B 0.000,C 180.000} C_DIS
LIN {X 76.380,Y 84.911,Z 59.027,A 180.000,B 0.000,C 180.000} C_DIS
LIN {X 76.069,Y 84.860,Z 59.022,A 180.000,B 0.000,C 180.000} C_DIS
LIN {X 75.762,Y 84.791,Z 59.018,A 180.000,B 0.000,C 180.000} C_DIS
LIN {X 75.457,Y 84.711,Z 59.014,A 180.000,B 0.000,C 180.000} C_DIS
LIN {X 75.155,Y 84.622,Z 59.011,A 180.000,B 0.000,C 180.000} C_DIS
LIN {X 74.859,Y 84.515,Z 59.008,A 180.000,B 0.000,C 180.000} C_DIS
LIN {X 74.567,Y 84.397,Z 59.005,A 180.000,B 0.000,C 180.000} C_DIS
LIN {X 74.278,Y 84.270,Z 59.003,A 180.000,B 0.000,C 180.000} C_DIS
LIN {X 73.998,Y 84.127,Z 59.002,A 180.000,B 0.000,C 180.000} C_DIS
LIN {X 73.723,Y 83.974,Z 59.001,A 180.000,B 0.000,C 180.000} C_DIS
LIN {X 73.453,Y 83.812,Z 59.000,A 180.000,B 0.000,C 180.000} C_DIS
LIN {X 73.260,Y 83.681,Z 59.000,A 180.000,B 0.000,C 180.000} C_DIS
; Cutting Move Starts
LIN {X 73.120,Y 83.586,Z 59.000,A 180.000,B 0.000,C 180.000} C_DIS
LIN {X 72.992,Y 83.489,Z 59.000,A 180.000,B 0.000,C 180.000} C_DIS
LIN {X 72.762,Y 83.310,Z 59.000,A 180.000,B 0.000,C 180.000} C_DIS
LIN {X 72.584,Y 83.158,Z 59.000,A 180.000,B 0.000,C 180.000} C_DIS
LIN {X 72.405,Y 83.000,Z 59.000,A 180.000,B 0.000,C 180.000} C_DIS
LIN {X 72.353,Y 82.952,Z 59.000,A 180.000,B 0.000,C 180.000} C_DIS
LIN {X 72.048,Y 82.647,Z 59.000,A 180.000,B 0.000,C 180.000} C_DIS
LIN {X 72.000,Y 82.595,Z 59.000,A 180.000,B 0.000,C 180.000} C_DIS
LIN {X 71.842,Y 82.416,Z 59.000,A 180.000,B 0.000,C 180.000} C_DIS
LIN {X 71.690,Y 82.238,Z 59.000,A 180.000,B 0.000,C 180.000} C_DIS
LIN {X 71.511,Y 82.008,Z 59.000,A 180.000,B 0.000,C 180.000} C_DIS
LIN {X 71.414,Y 81.880,Z 59.000,A 180.000,B 0.000,C 180.000} C_DIS
LIN {X 71.171,Y 81.522,Z 59.000,A 180.000,B 0.000,C 180.000} C_DIS
LIN {X 71.154,Y 81.493,Z 59.000,A 180.000,B 0.000,C 180.000} C_DIS
LIN {X 70.960,Y 81.165,Z 59.000,A 180.000,B 0.000,C 180.000} C_DIS
LIN {X 70.864,Y 80.986,Z 59.000,A 180.000,B 0.000,C 180.000} C_DIS
LIN {X 70.773,Y 80.807,Z 59.000,A 180.000,B 0.000,C 180.000} C_DIS
LIN {X 70.687,Y 80.628,Z 59.000,A 180.000,B 0.000,C 180.000} C_DIS
LIN {X 70.532,Y 80.271,Z 59.000,A 180.000,B 0.000,C 180.000} C_DIS
